LIN {X 0,Y 232.511,Z 383.184,A -85,B 0,C 180,E1 -19720.449,E2 -19720.449} C_VEL
LIN {X 0,Y 232.464,Z 384.387,A -85,B 0,C 180,E1 -19722.217,E2 -19722.217} C_VEL
LIN {X 0,Y 232.571,Z 385.359,A -85,B 0,C 180,E1 -19724.771,E2 -19724.771} C_VEL
LIN {X 0,Y 232.799,Z 385.455,A -85,B 0,C 180,E1 -19727.571,E2 -19727.571} C_VEL
LIN {X 0,Y 233.183,Z 384.978,A -85,B 0,C 180,E1 -19729.361,E2 -19729.361} C_VEL
LIN {X 0,Y 233.739,Z 384.005,A -85,B 0,C 180,E1 -19731.243,E2 -19731.243} C_VEL
LIN {X 0,Y 234.317,Z 382.734,A -85,B 0,C 180,E1 -19732.949,E2 -19732.949} C_VEL
LIN {X 0,Y 235.614,Z 379.876,A -85,B 0,C 180,E1 -19735.626,E2 -19735.626} C_VEL
LIN {X 0,Y 237.292,Z 375.916,A -85,B 0,C 180,E1 -19738.286,E2 -19738.286} C_VEL
LIN {X 0,Y 239.453,Z 370.738,A -85,B 0,C 180,E1 -19740.905,E2 -19740.905} C_VEL
LIN {X 0,Y 241.967,Z 364.116,A -85,B 0,C 180,E1 -19743.494,E2 -19743.494} C_VEL
LIN {X 0,Y 244.993,Z 355.784,A -85,B 0,C 180,E1 -19746.019,E2 -19746.019} C_VEL
LIN {X 0,Y 248.125,Z 346.362,A -85,B 0,C 180,E1 -19748.26,E2 -19748.26} C_VEL
LIN {X 0,Y 250.99,Z 336.548,A -85,B 0,C 180,E1 -19750.091,E2 -19750.091} C_VEL
LIN {X 0,Y 251.249,Z 333.713,A -85,B 0,C 180,E1 -19750.632,E2 -19750.632} C_VEL
LIN {X 0,Y 250.196,Z 324.296,A -85,B 0,C 180,E1 -19752.496,E2 -19752.496} C_VEL
LIN {X 0,Y 248.157,Z 314.273,A -85,B 0,C 180,E1 -19754.352,E2 -19754.352} C_VEL
LIN {X 0,Y 245.125,Z 303.736,A -85,B 0,C 180,E1 -19756.192,E2 -19756.192} C_VEL
LIN {X 0,Y 240.981,Z 293.088,A -85,B 0,C 180,E1 -19758.019,E2 -19758.019} C_VEL
LIN {X 0,Y 237.615,Z 286.034,A -85,B 0,C 180,E1 -19759.239,E2 -19759.239} C_VEL
LIN {X 0,Y 236.078,Z 283.158,A -85,B 0,C 180,E1 -19759.756,E2 -19759.756} C_VEL
LIN {X 0,Y 235.799,Z 281.871,A -85,B 0,C 180,E1 -19759.944,E2 -19759.944} C_VEL
LIN {X 0,Y 235.684,Z 279.573,A -85,B 0,C 180,E1 -19763.621,E2 -19763.621} C_VEL
LIN {X 0,Y 235.395,Z 277.379,A -85,B 0,C 180,E1 -19767.495,E2 -19767.495} C_VEL
LIN {X 0,Y 235.12,Z 275.354,A -85,B 0,C 180,E1 -19771.431,E2 -19771.431} C_VEL
LIN {X 0,Y 234.989,Z 274.23,A -85,B 0,C 180,E1 -19773.794,E2 -19773.794} C_VEL
LIN {X 0,Y 235.036,Z 274.205,A -85,B 0,C 180,E1 -19778.975,E2 -19778.975} C_VEL
LIN {X 0,Y 235.109,Z 274.195,A -85,B 0,C 180,E1 -19783.045,E2 -19783.045} C_VEL
LIN {X 0,Y 235.106,Z 274.199,A -85,B 0,C 180,E1 -19787.924,E2 -19787.924} C_VEL
LIN {X 0,Y 235.324,Z 274.172,A -85,B 0,C 180,E1 -19791.414,E2 -19791.414} C_VEL
LIN {X 0,Y 235.367,Z 274.166,A -85,B 0,C 180,E1 -19793.142,E2 -19793.142} C_VEL
LIN {X 0,Y 235.59,Z 274.14,A -85,B 0,C 180,E1 -19798.293,E2 -19798.293} C_VEL
LIN {X 0,Y 235.59,Z 274.138,A -85,B 0,C 180,E1 -19801.712,E2 -19801.712} C_VEL
LIN {X 0,Y 235.399,Z 274.164,A -85,B 0,C 180,E1 -19806.861,E2 -19806.861} C_VEL
LIN {X 0,Y 235.234,Z 274.184,A -85,B 0,C 180,E1 -19810.329,E2 -19810.329} C_VEL
LIN {X 0,Y 235.109,Z 274.201,A -85,B 0,C 180,E1 -19815.609,E2 -19815.609} C_VEL
LIN {X 0,Y 235.006,Z 274.216,A -85,B 0,C 180,E1 -19819.208,E2 -19819.208} C_VEL
LIN {X 0,Y 234.95,Z 274.225,A -85,B 0,C 180,E1 -19822.886,E2 -19822.886} C_VEL
LIN {X 0,Y 234.954,Z 274.225,A -85,B 0,C 180,E1 -19826.661,E2 -19826.661} C_VEL
LIN {X 0,Y 234.951,Z 274.386,A -85,B 0,C 180,E1 -19829.837,E2 -19829.837} C_VEL
LIN {X 0,Y 235.421,Z 276.965,A -85,B 0,C 180,E1 -19834.558,E2 -19834.558} C_VEL
LIN {X 0,Y 235.9,Z 279.582,A -85,B 0,C 180,E1 -19838.731,E2 -19838.731} C_VEL
LIN {X 0,Y 236.351,Z 282.705,A -85,B 0,C 180,E1 -19843.153,E2 -19843.153} C_VEL
LIN {X 0,Y 236.928,Z 286.376,A -85,B 0,C 180,E1 -19847.868,E2 -19847.868} C_VEL
LIN {X 0,Y 237.196,Z 289.485,A -85,B 0,C 180,E1 -19851.499,E2 -19851.499} C_VEL
LIN {X 0,Y 237.272,Z 290.986,A -85,B 0,C 180,E1 -19852.337,E2 -19852.337} C_VEL
LIN {X 0,Y 237.343,Z 293.485,A -85,B 0,C 180,E1 -19853.038,E2 -19853.038} C_VEL
LIN {X 0,Y 237.459,Z 298.336,A -85,B 0,C 180,E1 -19853.861,E2 -19853.861} C_VEL
LIN {X 0,Y 238.604,Z 313.774,A -85,B 0,C 180,E1 -19855.558,E2 -19855.558} C_VEL
LIN {X 0,Y 238.921,Z 315.576,A -85,B 0,C 180,E1 -19855.823,E2 -19855.823} C_VEL
LIN {X 0,Y 241.212,Z 326.613,A -85,B 0,C 180,E1 -19857.669,E2 -19857.669} C_VEL
LIN {X 0,Y 242.552,Z 337.882,A -85,B 0,C 180,E1 -19859.696,E2 -19859.696} C_VEL
LIN {X 0,Y 242.79,Z 347.643,A -85,B 0,C 180,E1 -19861.611,E2 -19861.611} C_VEL
LIN {X 0,Y 242.31,Z 353.451,A -85,B 0,C 180,E1 -19862.819,E2 -19862.819} C_VEL
LIN {X 0,Y 239.085,Z 362.778,A -85,B 0,C 180,E1 -19864.772,E2 -19864.772} C_VEL
LIN {X 0,Y 235.788,Z 371.794,A -85,B 0,C 180,E1 -19867.203,E2 -19867.203} C_VEL
LIN {X 0,Y 233.117,Z 379.081,A -85,B 0,C 180,E1 -19869.715,E2 -19869.715} C_VEL
LIN {X 0,Y 230.807,Z 384.952,A -85,B 0,C 180,E1 -19872.273,E2 -19872.273} C_VEL
LIN {X 0,Y 228.783,Z 389.609,A -85,B 0,C 180,E1 -19874.864,E2 -19874.864} C_VEL
LIN {X 0,Y 227.416,Z 393.183,A -85,B 0,C 180,E1 -19877.507,E2 -19877.507} C_VEL
LIN {X 0,Y 226.707,Z 395.036,A -85,B 0,C 180,E1 -19879.281,E2 -19879.281} C_VEL
LIN {X 0,Y 225.835,Z 397.451,A -85,B 0,C 180,E1 -19882.85,E2 -19882.85} C_VEL
LIN {X 0,Y 225.588,Z 398.332,A -85,B 0,C 180,E1 -19886.428,E2 -19886.428} C_VEL
LIN {X 0,Y 225.66,Z 398.156,A -85,B 0,C 180,E1 -19888.215,E2 -19888.215} C_VEL
LIN {X 0,Y 225.758,Z 397.585,A -85,B 0,C 180,E1 -19890,E2 -19890} C_VEL
LIN {X 0,Y 225.693,Z 396.616,A -85,B 0,C 180,E1 -19891.784,E2 -19891.784} C_VEL
LIN {X 0,Y 225.669,Z 394.1,A -85,B 0,C 180,E1 -19894.724,E2 -19894.724} C_VEL
LIN {X 0,Y 225.836,Z 391.102,A -85,B 0,C 180,E1 -19897.151,E2 -19897.151} C_VEL
LIN {X 0,Y 226.28,Z 386.756,A -85,B 0,C 180,E1 -19899.836,E2 -19899.836} C_VEL
LIN {X 0,Y 227.026,Z 381.193,A -85,B 0,C 180,E1 -19902.515,E2 -19902.515} C_VEL
LIN {X 0,Y 228.257,Z 374.239,A -85,B 0,C 180,E1 -19905.171,E2 -19905.171} C_VEL
LIN {X 0,Y 229.94,Z 365.512,A -85,B 0,C 180,E1 -19907.797,E2 -19907.797} C_VEL
LIN {X 0,Y 231.048,Z 358.488,A -85,B 0,C 180,E1 -19909.548,E2 -19909.548} C_VEL
LIN {X 0,Y 232.955,Z 347.829,A -85,B 0,C 180,E1 -19911.689,E2 -19911.689} C_VEL
LIN {X 0,Y 233.808,Z 341.483,A -85,B 0,C 180,E1 -19912.768,E2 -19912.768} C_VEL
LIN {X 0,Y 233.356,Z 330.679,A -85,B 0,C 180,E1 -19914.434,E2 -19914.434} C_VEL
LIN {X 0,Y 232.284,Z 318.675,A -85,B 0,C 180,E1 -19915.952,E2 -19915.952} C_VEL
LIN {X 0,Y 230.552,Z 306.518,A -85,B 0,C 180,E1 -19917.209,E2 -19917.209} C_VEL
LIN {X 0,Y 227.885,Z 293.983,A -85,B 0,C 180,E1 -19918.266,E2 -19918.266} C_VEL
LIN {X 0,Y 227.536,Z 291.964,A -85,B 0,C 180,E1 -19918.428,E2 -19918.428} C_VEL
LIN {X 0,Y 228.68,Z 286.481,A -85,B 0,C 180,E1 -19923.585,E2 -19923.585} C_VEL
LIN {X 0,Y 229.087,Z 284.326,A -85,B 0,C 180,E1 -19925.653,E2 -19925.653} C_VEL
LIN {X 0,Y 229.162,Z 282.142,A -85,B 0,C 180,E1 -19927.832,E2 -19927.832} C_VEL
LIN {X 0,Y 228.391,Z 277.71,A -85,B 0,C 180,E1 -19932.607,E2 -19932.607} C_VEL
LIN {X 0,Y 227.881,Z 275.105,A -85,B 0,C 180,E1 -19935.681,E2 -19935.681} C_VEL
LIN {X 0,Y 227.828,Z 275.111,A -85,B 0,C 180,E1 -19940.46,E2 -19940.46} C_VEL
LIN {X 0,Y 227.865,Z 275.102,A -85,B 0,C 180,E1 -19944.123,E2 -19944.123} C_VEL
LIN {X 0,Y 227.855,Z 275.103,A -85,B 0,C 180,E1 -19948.373,E2 -19948.373} C_VEL
LIN {X 0,Y 227.853,Z 275.103,A -85,B 0,C 180,E1 -19952.439,E2 -19952.439} C_VEL
LIN {X 0,Y 227.893,Z 275.095,A -85,B 0,C 180,E1 -19956.363,E2 -19956.363} C_VEL
LIN {X 0,Y 227.931,Z 275.095,A -85,B 0,C 180,E1 -19960.171,E2 -19960.171} C_VEL
LIN {X 0,Y 228.051,Z 275.076,A -85,B 0,C 180,E1 -19963.895,E2 -19963.895} C_VEL
LIN {X 0,Y 228.068,Z 275.075,A -85,B 0,C 180,E1 -19967.541,E2 -19967.541} C_VEL
LIN {X 0,Y 228.264,Z 275.05,A -85,B 0,C 180,E1 -19971.142,E2 -19971.142} C_VEL
LIN {X 0,Y 228.32,Z 275.044,A -85,B 0,C 180,E1 -19972.925,E2 -19972.925} C_VEL
LIN {X 0,Y 228.549,Z 274.995,A -85,B 0,C 180,E1 -19978.236,E2 -19978.236} C_VEL
LIN {X 0,Y 228.55,Z 275.004,A -85,B 0,C 180,E1 -19981.76,E2 -19981.76} C_VEL
LIN {X 0,Y 228.349,Z 275.04,A -85,B 0,C 180,E1 -19987.069,E2 -19987.069} C_VEL
LIN {X 0,Y 228.153,Z 275.06,A -85,B 0,C 180,E1 -19990.649,E2 -19990.649} C_VEL
LIN {X 0,Y 228.053,Z 275.076,A -85,B 0,C 180,E1 -19994.27,E2 -19994.27} C_VEL
LIN {X 0,Y 227.996,Z 275.082,A -85,B 0,C 180,E1 -19997.951,E2 -19997.951} C_VEL
LIN {X 0,Y 227.923,Z 275.09,A -85,B 0,C 180,E1 -20002.327,E2 -20002.327} C_VEL
LIN {X 0,Y 227.935,Z 275.09,A -85,B 0,C 180,E1 -20006.601,E2 -20006.601} C_VEL
LIN {X 0,Y 227.901,Z 275.089,A -85,B 0,C 180,E1 -20010.294,E2 -20010.294} C_VEL
LIN {X 0,Y 227.881,Z 275.096,A -85,B 0,C 180,E1 -20013.717,E2 -20013.717} C_VEL
LIN {X 0,Y 227.863,Z 275.097,A -85,B 0,C 180,E1 -20018.084,E2 -20018.084} C_VEL
LIN {X 0,Y 227.907,Z 275.091,A -85,B 0,C 180,E1 -20022.717,E2 -20022.717} C_VEL
LIN {X 0,Y 227.808,Z 275.103,A -85,B 0,C 180,E1 -20027.258,E2 -20027.258} C_VEL
LIN {X 0,Y 227.84,Z 275.102,A -85,B 0,C 180,E1 -20031.909,E2 -20031.909} C_VEL
LIN {X 0,Y 227.88,Z 275.1,A -85,B 0,C 180,E1 -20036.281,E2 -20036.281} C_VEL
LIN {X 0,Y 227.89,Z 275.099,A -85,B 0,C 180,E1 -20040.434,E2 -20040.434} C_VEL
LIN {X 0,Y 227.869,Z 275.103,A -85,B 0,C 180,E1 -20044.419,E2 -20044.419} C_VEL
LIN {X 0,Y 227.96,Z 275.126,A -85,B 0,C 180,E1 -20047.113,E2 -20047.113} C_VEL
LIN {X 0,Y 227.616,Z 277.511,A -85,B 0,C 180,E1 -20050.145,E2 -20050.145} C_VEL
LIN {X 0,Y 227.294,Z 281.12,A -85,B 0,C 180,E1 -20054.677,E2 -20054.677} C_VEL
LIN {X 0,Y 230.775,Z 294.117,A -85,B 0,C 180,E1 -20055.843,E2 -20055.843} C_VEL
LIN {X 0,Y 233.292,Z 305.864,A -85,B 0,C 180,E1 -20057.142,E2 -20057.142} C_VEL
LIN {X 0,Y 234.888,Z 316.795,A -85,B 0,C 180,E1 -20058.567,E2 -20058.567} C_VEL
LIN {X 0,Y 235.473,Z 324.331,A -85,B 0,C 180,E1 -20059.684,E2 -20059.684} C_VEL
LIN {X 0,Y 233.643,Z 334.908,A -85,B 0,C 180,E1 -20061.35,E2 -20061.35} C_VEL
LIN {X 0,Y 232.151,Z 343.57,A -85,B 0,C 180,E1 -20063.045,E2 -20063.045} C_VEL
LIN {X 0,Y 230.463,Z 352.528,A -85,B 0,C 180,E1 -20065.189,E2 -20065.189} C_VEL
LIN {X 0,Y 228.831,Z 361.274,A -85,B 0,C 180,E1 -20067.8,E2 -20067.8} C_VEL
LIN {X 0,Y 227.567,Z 368.252,A -85,B 0,C 180,E1 -20070.442,E2 -20070.442} C_VEL
LIN {X 0,Y 226.56,Z 374.651,A -85,B 0,C 180,E1 -20073.557,E2 -20073.557} C_VEL
LIN {X 0,Y 226.106,Z 378.454,A -85,B 0,C 180,E1 -20075.956,E2 -20075.956} C_VEL
LIN {X 0,Y 225.564,Z 382.022,A -85,B 0,C 180,E1 -20078.962,E2 -20078.962} C_VEL
LIN {X 0,Y 225.387,Z 383.598,A -85,B 0,C 180,E1 -20080.783,E2 -20080.783} C_VEL
LIN {X 0,Y 225.386,Z 384.708,A -85,B 0,C 180,E1 -20082.607,E2 -20082.607} C_VEL
LIN {X 0,Y 225.471,Z 385.548,A -85,B 0,C 180,E1 -20084.932,E2 -20084.932} C_VEL
LIN {X 0,Y 225.795,Z 385.622,A -85,B 0,C 180,E1 -20088.134,E2 -20088.134} C_VEL
LIN {X 0,Y 226.731,Z 384.25,A -85,B 0,C 180,E1 -20091.586,E2 -20091.586} C_VEL
LIN {X 0,Y 227.507,Z 382.724,A -85,B 0,C 180,E1 -20093.677,E2 -20093.677} C_VEL
LIN {X 0,Y 228.959,Z 379.765,A -85,B 0,C 180,E1 -20096.428,E2 -20096.428} C_VEL
LIN {X 0,Y 230.774,Z 375.692,A -85,B 0,C 180,E1 -20099.16,E2 -20099.16} C_VEL
LIN {X 0,Y 233.497,Z 369.324,A -85,B 0,C 180,E1 -20102.292,E2 -20102.292} C_VEL
LIN {X 0,Y 236.311,Z 362.316,A -85,B 0,C 180,E1 -20104.924,E2 -20104.924} C_VEL
LIN {X 0,Y 238.952,Z 355.344,A -85,B 0,C 180,E1 -20106.997,E2 -20106.997} C_VEL
LIN {X 0,Y 242.083,Z 346.319,A -85,B 0,C 180,E1 -20109.155,E2 -20109.155} C_VEL
LIN {X 0,Y 244.7,Z 337.791,A -85,B 0,C 180,E1 -20110.797,E2 -20110.797} C_VEL
LIN {X 0,Y 244.869,Z 335.253,A -85,B 0,C 180,E1 -20111.308,E2 -20111.308} C_VEL
LIN {X 0,Y 243.908,Z 325.616,A -85,B 0,C 180,E1 -20113.322,E2 -20113.322} C_VEL
LIN {X 0,Y 241.747,Z 314.782,A -85,B 0,C 180,E1 -20115.439,E2 -20115.439} C_VEL
LIN {X 0,Y 238.549,Z 304.085,A -85,B 0,C 180,E1 -20117.436,E2 -20117.436} C_VEL
LIN {X 0,Y 234.502,Z 293.899,A -85,B 0,C 180,E1 -20119.322,E2 -20119.322} C_VEL
LIN {X 0,Y 232.592,Z 290.047,A -85,B 0,C 180,E1 -20120.063,E2 -20120.063} C_VEL
LIN {X 0,Y 230.784,Z 286.427,A -85,B 0,C 180,E1 -20120.746,E2 -20120.746} C_VEL
LIN {X 0,Y 229.169,Z 283.393,A -85,B 0,C 180,E1 -20121.332,E2 -20121.332} C_VEL
LIN {X 0,Y 228.818,Z 282.124,A -85,B 0,C 180,E1 -20121.543,E2 -20121.543} C_VEL
LIN {X 0,Y 228.525,Z 279.364,A -85,B 0,C 180,E1 -20126.391,E2 -20126.391} C_VEL
LIN {X 0,Y 228.252,Z 277.253,A -85,B 0,C 180,E1 -20130.488,E2 -20130.488} C_VEL
LIN {X 0,Y 227.977,Z 275.452,A -85,B 0,C 180,E1 -20134.434,E2 -20134.434} C_VEL
LIN {X 0,Y 227.999,Z 275.086,A -85,B 0,C 180,E1 -20138.293,E2 -20138.293} C_VEL
LIN {X 0,Y 228.038,Z 275.075,A -85,B 0,C 180,E1 -20142.819,E2 -20142.819} C_VEL
LIN {X 0,Y 228.064,Z 275.077,A -85,B 0,C 180,E1 -20147.545,E2 -20147.545} C_VEL
LIN {X 0,Y 228.261,Z 275.052,A -85,B 0,C 180,E1 -20151.147,E2 -20151.147} C_VEL
LIN {X 0,Y 228.317,Z 275.046,A -85,B 0,C 180,E1 -20152.93,E2 -20152.93} C_VEL
LIN {X 0,Y 228.549,Z 275.016,A -85,B 0,C 180,E1 -20158.24,E2 -20158.24} C_VEL
LIN {X 0,Y 228.549,Z 275.015,A -85,B 0,C 180,E1 -20161.764,E2 -20161.764} C_VEL
LIN {X 0,Y 228.35,Z 275.042,A -85,B 0,C 180,E1 -20167.074,E2 -20167.074} C_VEL
LIN {X 0,Y 228.16,Z 275.066,A -85,B 0,C 180,E1 -20170.653,E2 -20170.653} C_VEL
LIN {X 0,Y 228.059,Z 275.08,A -85,B 0,C 180,E1 -20174.274,E2 -20174.274} C_VEL
LIN {X 0,Y 228.001,Z 275.089,A -85,B 0,C 180,E1 -20177.956,E2 -20177.956} C_VEL
LIN {X 0,Y 227.915,Z 275.102,A -85,B 0,C 180,E1 -20182.323,E2 -20182.323} C_VEL
LIN {X 0,Y 227.931,Z 275.1,A -85,B 0,C 180,E1 -20186.599,E2 -20186.599} C_VEL
LIN {X 0,Y 227.864,Z 275.107,A -85,B 0,C 180,E1 -20187.56,E2 -20187.56} C_VEL
LIN {X 0,Y 228.066,Z 276.286,A -85,B 0,C 180,E1 -20190.366,E2 -20190.366} C_VEL
LIN {X 0,Y 228.42,Z 278.112,A -85,B 0,C 180,E1 -20193.828,E2 -20193.828} C_VEL
LIN {X 0,Y 228.828,Z 280.553,A -85,B 0,C 180,E1 -20197.901,E2 -20197.901} C_VEL
LIN {X 0,Y 229.332,Z 283.544,A -85,B 0,C 180,E1 -20202.394,E2 -20202.394} C_VEL
LIN {X 0,Y 229.924,Z 287.556,A -85,B 0,C 180,E1 -20207.744,E2 -20207.744} C_VEL
LIN {X 0,Y 230.202,Z 290.962,A -85,B 0,C 180,E1 -20211.816,E2 -20211.816} C_VEL
LIN {X 0,Y 231.361,Z 294.432,A -85,B 0,C 180,E1 -20212.347,E2 -20212.347} C_VEL
LIN {X 0,Y 232.509,Z 296.395,A -85,B 0,C 180,E1 -20212.734,E2 -20212.734} C_VEL
LIN {X 0,Y 236.743,Z 307.783,A -85,B 0,C 180,E1 -20214.574,E2 -20214.574} C_VEL
LIN {X 0,Y 238.921,Z 315.576,A -85,B 0,C 180,E1 -20215.823,E2 -20215.823} C_VEL
LIN {X 0,Y 239.435,Z 320.71,A -85,B 0,C 180,E1 -20216.542,E2 -20216.542} C_VEL
LIN {X 0,Y 238.405,Z 329.615,A -85,B 0,C 180,E1 -20217.616,E2 -20217.616} C_VEL
LIN {X 0,Y 237.088,Z 336.477,A -85,B 0,C 180,E1 -20218.53,E2 -20218.53} C_VEL
LIN {X 0,Y 236.499,Z 341.335,A -85,B 0,C 180,E1 -20219.337,E2 -20219.337} C_VEL
LIN {X 0,Y 236.473,Z 342.85,A -85,B 0,C 180,E1 -20219.636,E2 -20219.636} C_VEL
LIN {X 0,Y 236.193,Z 352.965,A -85,B 0,C 180,E1 -20221.813,E2 -20221.813} C_VEL
LIN {X 0,Y 234.024,Z 359.687,A -85,B 0,C 180,E1 -20223.227,E2 -20223.227} C_VEL
LIN {X 0,Y 230.92,Z 367.846,A -85,B 0,C 180,E1 -20225.262,E2 -20225.262} C_VEL
LIN {X 0,Y 227.819,Z 375.722,A -85,B 0,C 180,E1 -20227.744,E2 -20227.744} C_VEL
LIN {X 0,Y 225.604,Z 381.322,A -85,B 0,C 180,E1 -20229.961,E2 -20229.961} C_VEL
LIN {X 0,Y 223.256,Z 386.696,A -85,B 0,C 180,E1 -20232.6,E2 -20232.6} C_VEL
LIN {X 0,Y 221.326,Z 390.916,A -85,B 0,C 180,E1 -20235.284,E2 -20235.284} C_VEL
LIN {X 0,Y 220.458,Z 393.166,A -85,B 0,C 180,E1 -20237.106,E2 -20237.106} C_VEL
LIN {X 0,Y 219.712,Z 394.964,A -85,B 0,C 180,E1 -20238.935,E2 -20238.935} C_VEL
LIN {X 0,Y 218.792,Z 397.319,A -85,B 0,C 180,E1 -20242.618,E2 -20242.618} C_VEL
LIN {X 0,Y 218.489,Z 398.087,A -85,B 0,C 180,E1 -20245.702,E2 -20245.702} C_VEL
LIN {X 0,Y 218.575,Z 397.915,A -85,B 0,C 180,E1 -20248.158,E2 -20248.158} C_VEL
LIN {X 0,Y 218.671,Z 397.316,A -85,B 0,C 180,E1 -20250,E2 -20250} C_VEL
LIN {X 0,Y 218.589,Z 396.318,A -85,B 0,C 180,E1 -20251.843,E2 -20251.843} C_VEL
LIN {X 0,Y 218.581,Z 394.005,A -85,B 0,C 180,E1 -20254.61,E2 -20254.61} C_VEL
LIN {X 0,Y 218.788,Z 390.687,A -85,B 0,C 180,E1 -20257.382,E2 -20257.382} C_VEL
LIN {X 0,Y 219.269,Z 386.275,A -85,B 0,C 180,E1 -20260.153,E2 -20260.153} C_VEL
LIN {X 0,Y 220.036,Z 380.639,A -85,B 0,C 180,E1 -20262.919,E2 -20262.919} C_VEL
LIN {X 0,Y 221.384,Z 373.593,A -85,B 0,C 180,E1 -20265.654,E2 -20265.654} C_VEL
LIN {X 0,Y 223.125,Z 364.74,A -85,B 0,C 180,E1 -20268.359,E2 -20268.359} C_VEL
LIN {X 0,Y 224.085,Z 358.762,A -85,B 0,C 180,E1 -20269.897,E2 -20269.897} C_VEL
LIN {X 0,Y 225.832,Z 349.17,A -85,B 0,C 180,E1 -20271.928,E2 -20271.928} C_VEL
LIN {X 0,Y 226.917,Z 343.013,A -85,B 0,C 180,E1 -20273.017,E2 -20273.017} C_VEL
LIN {X 0,Y 226.553,Z 331.665,A -85,B 0,C 180,E1 -20274.875,E2 -20274.875} C_VEL
LIN {X 0,Y 225.576,Z 319.872,A -85,B 0,C 180,E1 -20276.461,E2 -20276.461} C_VEL
LIN {X 0,Y 223.926,Z 307.765,A -85,B 0,C 180,E1 -20277.789,E2 -20277.789} C_VEL
LIN {X 0,Y 221.22,Z 294.742,A -85,B 0,C 180,E1 -20278.956,E2 -20278.956} C_VEL
LIN {X 0,Y 220.581,Z 291.788,A -85,B 0,C 180,E1 -20279.206,E2 -20279.206} C_VEL
LIN {X 0,Y 221.383,Z 288.221,A -85,B 0,C 180,E1 -20282.661,E2 -20282.661} C_VEL
LIN {X 0,Y 222.043,Z 284.998,A -85,B 0,C 180,E1 -20285.841,E2 -20285.841} C_VEL
LIN {X 0,Y 222.143,Z 283.177,A -85,B 0,C 180,E1 -20287.724,E2 -20287.724} C_VEL
LIN {X 0,Y 221.501,Z 279.503,A -85,B 0,C 180,E1 -20291.782,E2 -20291.782} C_VEL
LIN {X 0,Y 220.83,Z 275.983,A -85,B 0,C 180,E1 -20295.983,E2 -20295.983} C_VEL
LIN {X 0,Y 220.782,Z 275.989,A -85,B 0,C 180,E1 -20300.456,E2 -20300.456} C_VEL
LIN {X 0,Y 220.826,Z 275.982,A -85,B 0,C 180,E1 -20302.791,E2 -20302.791} C_VEL
LIN {X 0,Y 220.812,Z 275.979,A -85,B 0,C 180,E1 -20307.241,E2 -20307.241} C_VEL
LIN {X 0,Y 220.803,Z 275.978,A -85,B 0,C 180,E1 -20311.479,E2 -20311.479} C_VEL
LIN {X 0,Y 220.846,Z 275.971,A -85,B 0,C 180,E1 -20315.56,E2 -20315.56} C_VEL
LIN {X 0,Y 220.882,Z 275.971,A -85,B 0,C 180,E1 -20319.511,E2 -20319.511} C_VEL
LIN {X 0,Y 221.012,Z 275.952,A -85,B 0,C 180,E1 -20323.368,E2 -20323.368} C_VEL
LIN {X 0,Y 221.064,Z 275.943,A -85,B 0,C 180,E1 -20329.001,E2 -20329.001} C_VEL
LIN {X 0,Y 221.255,Z 275.924,A -85,B 0,C 180,E1 -20332.698,E2 -20332.698} C_VEL
LIN {X 0,Y 221.507,Z 275.871,A -85,B 0,C 180,E1 -20338.18,E2 -20338.18} C_VEL
LIN {X 0,Y 221.508,Z 275.88,A -85,B 0,C 180,E1 -20341.816,E2 -20341.816} C_VEL
LIN {X 0,Y 221.3,Z 275.919,A -85,B 0,C 180,E1 -20347.296,E2 -20347.296} C_VEL
LIN {X 0,Y 221.101,Z 275.939,A -85,B 0,C 180,E1 -20350.992,E2 -20350.992} C_VEL
LIN {X 0,Y 221.008,Z 275.948,A -85,B 0,C 180,E1 -20356.628,E2 -20356.628} C_VEL
LIN {X 0,Y 220.885,Z 275.969,A -85,B 0,C 180,E1 -20360.484,E2 -20360.484} C_VEL
LIN {X 0,Y 220.86,Z 275.967,A -85,B 0,C 180,E1 -20364.433,E2 -20364.433} C_VEL
LIN {X 0,Y 220.829,Z 275.974,A -85,B 0,C 180,E1 -20368.512,E2 -20368.512} C_VEL
LIN {X 0,Y 220.816,Z 275.977,A -85,B 0,C 180,E1 -20372.753,E2 -20372.753} C_VEL
LIN {X 0,Y 220.83,Z 275.973,A -85,B 0,C 180,E1 -20377.286,E2 -20377.286} C_VEL
LIN {X 0,Y 220.851,Z 275.969,A -85,B 0,C 180,E1 -20381.93,E2 -20381.93} C_VEL
LIN {X 0,Y 220.779,Z 275.982,A -85,B 0,C 180,E1 -20385.548,E2 -20385.548} C_VEL
LIN {X 0,Y 220.798,Z 275.982,A -85,B 0,C 180,E1 -20390.462,E2 -20390.462} C_VEL
LIN {X 0,Y 220.815,Z 275.977,A -85,B 0,C 180,E1 -20392.792,E2 -20392.792} C_VEL
LIN {X 0,Y 220.813,Z 275.979,A -85,B 0,C 180,E1 -20397.244,E2 -20397.244} C_VEL
LIN {X 0,Y 220.807,Z 275.979,A -85,B 0,C 180,E1 -20401.483,E2 -20401.483} C_VEL
LIN {X 0,Y 220.84,Z 275.978,A -85,B 0,C 180,E1 -20405.562,E2 -20405.562} C_VEL
LIN {X 0,Y 220.917,Z 276.039,A -85,B 0,C 180,E1 -20407.016,E2 -20407.016} C_VEL
LIN {X 0,Y 220.43,Z 279.415,A -85,B 0,C 180,E1 -20411.408,E2 -20411.408} C_VEL
LIN {X 0,Y 220.298,Z 281.3,A -85,B 0,C 180,E1 -20413.851,E2 -20413.851} C_VEL
LIN {X 0,Y 224.497,Z 296.96,A -85,B 0,C 180,E1 -20415.4,E2 -20415.4} C_VEL
LIN {X 0,Y 226.85,Z 308.464,A -85,B 0,C 180,E1 -20416.772,E2 -20416.772} C_VEL
LIN {X 0,Y 228.236,Z 318.903,A -85,B 0,C 180,E1 -20418.229,E2 -20418.229} C_VEL
LIN {X 0,Y 228.726,Z 324.731,A -85,B 0,C 180,E1 -20419.152,E2 -20419.152} C_VEL
LIN {X 0,Y 226.83,Z 335.274,A -85,B 0,C 180,E1 -20420.863,E2 -20420.863} C_VEL
LIN {X 0,Y 225.146,Z 344.875,A -85,B 0,C 180,E1 -20422.827,E2 -20422.827} C_VEL
LIN {X 0,Y 223.372,Z 353.659,A -85,B 0,C 180,E1 -20425.036,E2 -20425.036} C_VEL
LIN {X 0,Y 222.009,Z 360.89,A -85,B 0,C 180,E1 -20427.278,E2 -20427.278} C_VEL
LIN {X 0,Y 220.612,Z 368.018,A -85,B 0,C 180,E1 -20430,E2 -20430} C_VEL
LIN {X 0,Y 219.651,Z 373.692,A -85,B 0,C 180,E1 -20432.751,E2 -20432.751} C_VEL
LIN {X 0,Y 219.013,Z 378.657,A -85,B 0,C 180,E1 -20435.888,E2 -20435.888} C_VEL
LIN {X 0,Y 218.428,Z 382.484,A -85,B 0,C 180,E1 -20439.257,E2 -20439.257} C_VEL
LIN {X 0,Y 218.271,Z 383.978,A -85,B 0,C 180,E1 -20441.139,E2 -20441.139} C_VEL
LIN {X 0,Y 218.282,Z 385.029,A -85,B 0,C 180,E1 -20443.025,E2 -20443.025} C_VEL
LIN {X 0,Y 218.381,Z 385.739,A -85,B 0,C 180,E1 -20445.112,E2 -20445.112} C_VEL
LIN {X 0,Y 218.49,Z 385.951,A -85,B 0,C 180,E1 -20446.827,E2 -20446.827} C_VEL
LIN {X 0,Y 218.814,Z 385.758,A -85,B 0,C 180,E1 -20448.734,E2 -20448.734} C_VEL
LIN {X 0,Y 219.769,Z 384.479,A -85,B 0,C 180,E1 -20451.976,E2 -20451.976} C_VEL
LIN {X 0,Y 220.729,Z 382.683,A -85,B 0,C 180,E1 -20454.451,E2 -20454.451} C_VEL
LIN {X 0,Y 222.732,Z 378.734,A -85,B 0,C 180,E1 -20457.938,E2 -20457.938} C_VEL
LIN {X 0,Y 225.082,Z 373.767,A -85,B 0,C 180,E1 -20461.01,E2 -20461.01} C_VEL
LIN {X 0,Y 227.712,Z 367.864,A -85,B 0,C 180,E1 -20463.747,E2 -20463.747} C_VEL
LIN {X 0,Y 230.815,Z 360.387,A -85,B 0,C 180,E1 -20466.422,E2 -20466.422} C_VEL
LIN {X 0,Y 233.761,Z 352.744,A -85,B 0,C 180,E1 -20468.589,E2 -20468.589} C_VEL
LIN {X 0,Y 237.016,Z 343.361,A -85,B 0,C 180,E1 -20470.717,E2 -20470.717} C_VEL
LIN {X 0,Y 238.547,Z 338.428,A -85,B 0,C 180,E1 -20471.66,E2 -20471.66} C_VEL
LIN {X 0,Y 238.05,Z 330.485,A -85,B 0,C 180,E1 -20473.44,E2 -20473.44} C_VEL
LIN {X 0,Y 236.549,Z 320.835,A -85,B 0,C 180,E1 -20475.482,E2 -20475.482} C_VEL
LIN {X 0,Y 234.082,Z 310.774,A -85,B 0,C 180,E1 -20477.509,E2 -20477.509} C_VEL
LIN {X 0,Y 230.19,Z 299.404,A -85,B 0,C 180,E1 -20479.753,E2 -20479.753} C_VEL
LIN {X 0,Y 226.034,Z 290.791,A -85,B 0,C 180,E1 -20481.552,E2 -20481.552} C_VEL
LIN {X 0,Y 224.162,Z 287.123,A -85,B 0,C 180,E1 -20482.316,E2 -20482.316} C_VEL
LIN {X 0,Y 222.322,Z 284.357,A -85,B 0,C 180,E1 -20482.991,E2 -20482.991} C_VEL
LIN {X 0,Y 221.731,Z 282.416,A -85,B 0,C 180,E1 -20483.328,E2 -20483.328} C_VEL
LIN {X 0,Y 221.452,Z 280.252,A -85,B 0,C 180,E1 -20487.353,E2 -20487.353} C_VEL
LIN {X 0,Y 221.21,Z 278.217,A -85,B 0,C 180,E1 -20491.542,E2 -20491.542} C_VEL
LIN {X 0,Y 220.933,Z 276.491,A -85,B 0,C 180,E1 -20495.575,E2 -20495.575} C_VEL
LIN {X 0,Y 220.931,Z 275.962,A -85,B 0,C 180,E1 -20497.562,E2 -20497.562} C_VEL
LIN {X 0,Y 220.986,Z 275.952,A -85,B 0,C 180,E1 -20502.566,E2 -20502.566} C_VEL
LIN {X 0,Y 221.003,Z 275.958,A -85,B 0,C 180,E1 -20507.14,E2 -20507.14} C_VEL
LIN {X 0,Y 221.198,Z 275.933,A -85,B 0,C 180,E1 -20510.861,E2 -20510.861} C_VEL
LIN {X 0,Y 221.253,Z 275.927,A -85,B 0,C 180,E1 -20512.703,E2 -20512.703} C_VEL
LIN {X 0,Y 221.507,Z 275.893,A -85,B 0,C 180,E1 -20518.184,E2 -20518.184} C_VEL
LIN {X 0,Y 221.507,Z 275.892,A -85,B 0,C 180,E1 -20521.82,E2 -20521.82} C_VEL
LIN {X 0,Y 221.285,Z 275.921,A -85,B 0,C 180,E1 -20527.301,E2 -20527.301} C_VEL
LIN {X 0,Y 221.109,Z 275.944,A -85,B 0,C 180,E1 -20530.996,E2 -20530.996} C_VEL
LIN {X 0,Y 221.014,Z 275.96,A -85,B 0,C 180,E1 -20536.632,E2 -20536.632} C_VEL
LIN {X 0,Y 220.883,Z 275.977,A -85,B 0,C 180,E1 -20540.489,E2 -20540.489} C_VEL
LIN {X 0,Y 220.855,Z 275.981,A -85,B 0,C 180,E1 -20544.439,E2 -20544.439} C_VEL
LIN {X 0,Y 220.907,Z 276.372,A -85,B 0,C 180,E1 -20547.029,E2 -20547.029} C_VEL
LIN {X 0,Y 221.178,Z 278.178,A -85,B 0,C 180,E1 -20550.917,E2 -20550.917} C_VEL
LIN {X 0,Y 221.555,Z 280.238,A -85,B 0,C 180,E1 -20554.821,E2 -20554.821} C_VEL
LIN {X 0,Y 221.88,Z 281.874,A -85,B 0,C 180,E1 -20557.641,E2 -20557.641} C_VEL
LIN {X 0,Y 222.255,Z 284.431,A -85,B 0,C 180,E1 -20561.612,E2 -20561.612} C_VEL
LIN {X 0,Y 222.755,Z 287.926,A -85,B 0,C 180,E1 -20566.526,E2 -20566.526} C_VEL
LIN {X 0,Y 223.166,Z 290.957,A -85,B 0,C 180,E1 -20570.149,E2 -20570.149} C_VEL
LIN {X 0,Y 224.317,Z 294.058,A -85,B 0,C 180,E1 -20570.642,E2 -20570.642} C_VEL
LIN {X 0,Y 225.801,Z 296.531,A -85,B 0,C 180,E1 -20571.178,E2 -20571.178} C_VEL
LIN {X 0,Y 229.153,Z 304.463,A -85,B 0,C 180,E1 -20572.624,E2 -20572.624} C_VEL
LIN {X 0,Y 232.696,Z 316.012,A -85,B 0,C 180,E1 -20574.636,E2 -20574.636} C_VEL
LIN {X 0,Y 234.972,Z 327.305,A -85,B 0,C 180,E1 -20576.636,E2 -20576.636} C_VEL
LIN {X 0,Y 236.262,Z 338.849,A -85,B 0,C 180,E1 -20578.822,E2 -20578.822} C_VEL
LIN {X 0,Y 236.473,Z 342.85,A -85,B 0,C 180,E1 -20579.636,E2 -20579.636} C_VEL
LIN {X 0,Y 235.895,Z 346.01,A -85,B 0,C 180,E1 -20580.19,E2 -20580.19} C_VEL
LIN {X 0,Y 234.407,Z 349.2,A -85,B 0,C 180,E1 -20580.649,E2 -20580.649} C_VEL
LIN {X 0,Y 229.068,Z 357.351,A -85,B 0,C 180,E1 -20581.843,E2 -20581.843} C_VEL
LIN {X 0,Y 228.063,Z 359.319,A -85,B 0,C 180,E1 -20582.243,E2 -20582.243} C_VEL
LIN {X 0,Y 224.503,Z 368.177,A -85,B 0,C 180,E1 -20584.505,E2 -20584.505} C_VEL
LIN {X 0,Y 221.048,Z 376.463,A -85,B 0,C 180,E1 -20587.228,E2 -20587.228} C_VEL
LIN {X 0,Y 218.127,Z 383.379,A -85,B 0,C 180,E1 -20590.227,E2 -20590.227} C_VEL
LIN {X 0,Y 215.739,Z 388.279,A -85,B 0,C 180,E1 -20592.952,E2 -20592.952} C_VEL
LIN {X 0,Y 213.944,Z 392.081,A -85,B 0,C 180,E1 -20595.737,E2 -20595.737} C_VEL
LIN {X 0,Y 212.734,Z 394.889,A -85,B 0,C 180,E1 -20598.568,E2 -20598.568} C_VEL
LIN {X 0,Y 211.723,Z 397.188,A -85,B 0,C 180,E1 -20602.37,E2 -20602.37} C_VEL
LIN {X 0,Y 211.399,Z 397.925,A -85,B 0,C 180,E1 -20605.855,E2 -20605.855} C_VEL
LIN {X 0,Y 211.473,Z 397.672,A -85,B 0,C 180,E1 -20608.096,E2 -20608.096} C_VEL
LIN {X 0,Y 211.586,Z 397.047,A -85,B 0,C 180,E1 -20610,E2 -20610} C_VEL
LIN {X 0,Y 211.488,Z 396.02,A -85,B 0,C 180,E1 -20611.904,E2 -20611.904} C_VEL
LIN {X 0,Y 211.479,Z 393.962,A -85,B 0,C 180,E1 -20614.432,E2 -20614.432} C_VEL
LIN {X 0,Y 211.712,Z 390.269,A -85,B 0,C 180,E1 -20617.63,E2 -20617.63} C_VEL
LIN {X 0,Y 212.235,Z 385.792,A -85,B 0,C 180,E1 -20620.494,E2 -20620.494} C_VEL
LIN {X 0,Y 213.072,Z 380.085,A -85,B 0,C 180,E1 -20623.349,E2 -20623.349} C_VEL
LIN {X 0,Y 214.525,Z 372.922,A -85,B 0,C 180,E1 -20626.168,E2 -20626.168} C_VEL
LIN {X 0,Y 216.268,Z 363.961,A -85,B 0,C 180,E1 -20628.963,E2 -20628.963} C_VEL
LIN {X 0,Y 217.29,Z 358.378,A -85,B 0,C 180,E1 -20630.424,E2 -20630.424} C_VEL
LIN {X 0,Y 219.274,Z 348.158,A -85,B 0,C 180,E1 -20632.619,E2 -20632.619} C_VEL
LIN {X 0,Y 220.051,Z 343.203,A -85,B 0,C 180,E1 -20633.529,E2 -20633.529} C_VEL
LIN {X 0,Y 219.692,Z 331.703,A -85,B 0,C 180,E1 -20635.488,E2 -20635.488} C_VEL
LIN {X 0,Y 218.808,Z 320.335,A -85,B 0,C 180,E1 -20637.083,E2 -20637.083} C_VEL
LIN {X 0,Y 217.249,Z 308.688,A -85,B 0,C 180,E1 -20638.434,E2 -20638.434} C_VEL
LIN {X 0,Y 214.755,Z 296.536,A -85,B 0,C 180,E1 -20639.607,E2 -20639.607} C_VEL
LIN {X 0,Y 213.65,Z 291.628,A -85,B 0,C 180,E1 -20640.007,E2 -20640.007} C_VEL
LIN {X 0,Y 214.52,Z 287.821,A -85,B 0,C 180,E1 -20643.844,E2 -20643.844} C_VEL
LIN {X 0,Y 215.077,Z 284.632,A -85,B 0,C 180,E1 -20647.158,E2 -20647.158} C_VEL
LIN {X 0,Y 214.557,Z 281.124,A -85,B 0,C 180,E1 -20651.113,E2 -20651.113} C_VEL
LIN {X 0,Y 213.779,Z 276.862,A -85,B 0,C 180,E1 -20656.338,E2 -20656.338} C_VEL
LIN {X 0,Y 213.705,Z 276.869,A -85,B 0,C 180,E1 -20661.327,E2 -20661.327} C_VEL
LIN {X 0,Y 213.754,Z 276.858,A -85,B 0,C 180,E1 -20666.015,E2 -20666.015} C_VEL
LIN {X 0,Y 213.75,Z 276.856,A -85,B 0,C 180,E1 -20670.447,E2 -20670.447} C_VEL
LIN {X 0,Y 213.781,Z 276.854,A -85,B 0,C 180,E1 -20674.697,E2 -20674.697} C_VEL
LIN {X 0,Y 213.802,Z 276.854,A -85,B 0,C 180,E1 -20678.8,E2 -20678.8} C_VEL
LIN {X 0,Y 213.941,Z 276.833,A -85,B 0,C 180,E1 -20682.801,E2 -20682.801} C_VEL
LIN {X 0,Y 213.948,Z 276.834,A -85,B 0,C 180,E1 -20686.704,E2 -20686.704} C_VEL
LIN {X 0,Y 214.139,Z 276.811,A -85,B 0,C 180,E1 -20690.553,E2 -20690.553} C_VEL
LIN {X 0,Y 214.096,Z 276.814,A -85,B 0,C 180,E1 -20694.346,E2 -20694.346} C_VEL
LIN {X 0,Y 214.44,Z 276.75,A -85,B 0,C 180,E1 -20698.12,E2 -20698.12} C_VEL
LIN {X 0,Y 214.55,Z 276.735,A -85,B 0,C 180,E1 -20699.998,E2 -20699.998} C_VEL
LIN {X 0,Y 214.441,Z 276.76,A -85,B 0,C 180,E1 -20701.876,E2 -20701.876} C_VEL
LIN {X 0,Y 214.235,Z 276.8,A -85,B 0,C 180,E1 -20707.538,E2 -20707.538} C_VEL
LIN {X 0,Y 214.017,Z 276.823,A -85,B 0,C 180,E1 -20711.361,E2 -20711.361} C_VEL
LIN {X 0,Y 213.924,Z 276.837,A -85,B 0,C 180,E1 -20715.235,E2 -20715.235} C_VEL
LIN {X 0,Y 213.833,Z 276.848,A -85,B 0,C 180,E1 -20719.185,E2 -20719.185} C_VEL
LIN {X 0,Y 213.84,Z 276.843,A -85,B 0,C 180,E1 -20723.225,E2 -20723.225} C_VEL
LIN {X 0,Y 213.822,Z 276.849,A -85,B 0,C 180,E1 -20727.448,E2 -20727.448} C_VEL
LIN {X 0,Y 213.772,Z 276.853,A -85,B 0,C 180,E1 -20731.734,E2 -20731.734} C_VEL
LIN {X 0,Y 213.746,Z 276.853,A -85,B 0,C 180,E1 -20736.285,E2 -20736.285} C_VEL
LIN {X 0,Y 213.789,Z 276.851,A -85,B 0,C 180,E1 -20741.104,E2 -20741.104} C_VEL
LIN {X 0,Y 213.8,Z 276.85,A -85,B 0,C 180,E1 -20743.684,E2 -20743.684} C_VEL
LIN {X 0,Y 213.705,Z 276.863,A -85,B 0,C 180,E1 -20748.874,E2 -20748.874} C_VEL
LIN {X 0,Y 213.739,Z 276.858,A -85,B 0,C 180,E1 -20753.712,E2 -20753.712} C_VEL
LIN {X 0,Y 213.76,Z 276.859,A -85,B 0,C 180,E1 -20758.262,E2 -20758.262} C_VEL
LIN {X 0,Y 213.777,Z 276.858,A -85,B 0,C 180,E1 -20762.597,E2 -20762.597} C_VEL
LIN {X 0,Y 213.866,Z 276.97,A -85,B 0,C 180,E1 -20766.938,E2 -20766.938} C_VEL
LIN {X 0,Y 213.451,Z 279.828,A -85,B 0,C 180,E1 -20770.777,E2 -20770.777} C_VEL
LIN {X 0,Y 213.308,Z 281.533,A -85,B 0,C 180,E1 -20773.036,E2 -20773.036} C_VEL
LIN {X 0,Y 217.005,Z 294.785,A -85,B 0,C 180,E1 -20774.375,E2 -20774.375} C_VEL
LIN {X 0,Y 219.741,Z 307.348,A -85,B 0,C 180,E1 -20775.903,E2 -20775.903} C_VEL
LIN {X 0,Y 221.235,Z 317.768,A -85,B 0,C 180,E1 -20777.385,E2 -20777.385} C_VEL
LIN {X 0,Y 221.968,Z 325.141,A -85,B 0,C 180,E1 -20778.587,E2 -20778.587} C_VEL
LIN {X 0,Y 219.859,Z 336.805,A -85,B 0,C 180,E1 -20780.571,E2 -20780.571} C_VEL
LIN {X 0,Y 218.435,Z 344.245,A -85,B 0,C 180,E1 -20782.141,E2 -20782.141} C_VEL
LIN {X 0,Y 216.62,Z 353.158,A -85,B 0,C 180,E1 -20784.414,E2 -20784.414} C_VEL
LIN {X 0,Y 214.868,Z 361.854,A -85,B 0,C 180,E1 -20787.188,E2 -20787.188} C_VEL
LIN {X 0,Y 213.517,Z 368.792,A -85,B 0,C 180,E1 -20790,E2 -20790} C_VEL
LIN {X 0,Y 212.524,Z 374.355,A -85,B 0,C 180,E1 -20792.843,E2 -20792.843} C_VEL
LIN {X 0,Y 211.933,Z 378.904,A -85,B 0,C 180,E1 -20795.849,E2 -20795.849} C_VEL
LIN {X 0,Y 211.568,Z 381.048,A -85,B 0,C 180,E1 -20797.635,E2 -20797.635} C_VEL
LIN {X 0,Y 211.297,Z 382.935,A -85,B 0,C 180,E1 -20799.573,E2 -20799.573} C_VEL
LIN {X 0,Y 211.157,Z 384.345,A -85,B 0,C 180,E1 -20801.519,E2 -20801.519} C_VEL
LIN {X 0,Y 211.185,Z 385.351,A -85,B 0,C 180,E1 -20803.471,E2 -20803.471} C_VEL
LIN {X 0,Y 211.306,Z 385.962,A -85,B 0,C 180,E1 -20805.431,E2 -20805.431} C_VEL
LIN {X 0,Y 211.47,Z 386.144,A -85,B 0,C 180,E1 -20807.403,E2 -20807.403} C_VEL
LIN {X 0,Y 211.849,Z 385.893,A -85,B 0,C 180,E1 -20809.374,E2 -20809.374} C_VEL
LIN {X 0,Y 212.795,Z 384.719,A -85,B 0,C 180,E1 -20812.375,E2 -20812.375} C_VEL
LIN {X 0,Y 214.022,Z 382.626,A -85,B 0,C 180,E1 -20815.27,E2 -20815.27} C_VEL
LIN {X 0,Y 215.936,Z 379.038,A -85,B 0,C 180,E1 -20818.512,E2 -20818.512} C_VEL
LIN {X 0,Y 217.897,Z 375.16,A -85,B 0,C 180,E1 -20821.067,E2 -20821.067} C_VEL
LIN {X 0,Y 220.898,Z 368.907,A -85,B 0,C 180,E1 -20824.192,E2 -20824.192} C_VEL
LIN {X 0,Y 223.749,Z 362.556,A -85,B 0,C 180,E1 -20826.64,E2 -20826.64} C_VEL
LIN {X 0,Y 226.841,Z 355.038,A -85,B 0,C 180,E1 -20828.955,E2 -20828.955} C_VEL
LIN {X 0,Y 230.414,Z 345.462,A -85,B 0,C 180,E1 -20831.268,E2 -20831.268} C_VEL
LIN {X 0,Y 231.972,Z 340.907,A -85,B 0,C 180,E1 -20832.189,E2 -20832.189} C_VEL
LIN {X 0,Y 232.223,Z 337.736,A -85,B 0,C 180,E1 -20832.918,E2 -20832.918} C_VEL
LIN {X 0,Y 231.372,Z 328.347,A -85,B 0,C 180,E1 -20835.111,E2 -20835.111} C_VEL
LIN {X 0,Y 229.584,Z 318.493,A -85,B 0,C 180,E1 -20837.279,E2 -20837.279} C_VEL
LIN {X 0,Y 226.814,Z 308.521,A -85,B 0,C 180,E1 -20839.409,E2 -20839.409} C_VEL
LIN {X 0,Y 223.889,Z 300.538,A -85,B 0,C 180,E1 -20841.114,E2 -20841.114} C_VEL
LIN {X 0,Y 219.68,Z 291.959,A -85,B 0,C 180,E1 -20843.087,E2 -20843.087} C_VEL
LIN {X 0,Y 217.7,Z 288.265,A -85,B 0,C 180,E1 -20843.959,E2 -20843.959} C_VEL
LIN {X 0,Y 215.245,Z 284.675,A -85,B 0,C 180,E1 -20844.932,E2 -20844.932} C_VEL
LIN {X 0,Y 214.653,Z 282.705,A -85,B 0,C 180,E1 -20845.279,E2 -20845.279} C_VEL
LIN {X 0,Y 214.318,Z 280.131,A -85,B 0,C 180,E1 -20850.538,E2 -20850.538} C_VEL
LIN {X 0,Y 214.056,Z 278.343,A -85,B 0,C 180,E1 -20854.737,E2 -20854.737} C_VEL
LIN {X 0,Y 213.847,Z 276.845,A -85,B 0,C 180,E1 -20858.81,E2 -20858.81} C_VEL
LIN {X 0,Y 213.963,Z 276.827,A -85,B 0,C 180,E1 -20862.808,E2 -20862.808} C_VEL
LIN {X 0,Y 213.945,Z 276.833,A -85,B 0,C 180,E1 -20866.709,E2 -20866.709} C_VEL
LIN {X 0,Y 214.136,Z 276.812,A -85,B 0,C 180,E1 -20870.557,E2 -20870.557} C_VEL
LIN {X 0,Y 214.095,Z 276.817,A -85,B 0,C 180,E1 -20874.351,E2 -20874.351} C_VEL
LIN {X 0,Y 214.44,Z 276.773,A -85,B 0,C 180,E1 -20878.124,E2 -20878.124} C_VEL
LIN {X 0,Y 214.54,Z 276.759,A -85,B 0,C 180,E1 -20880.002,E2 -20880.002} C_VEL
LIN {X 0,Y 214.44,Z 276.772,A -85,B 0,C 180,E1 -20881.88,E2 -20881.88} C_VEL
LIN {X 0,Y 214.224,Z 276.799,A -85,B 0,C 180,E1 -20887.543,E2 -20887.543} C_VEL
LIN {X 0,Y 214.041,Z 276.823,A -85,B 0,C 180,E1 -20891.364,E2 -20891.364} C_VEL
LIN {X 0,Y 213.929,Z 276.839,A -85,B 0,C 180,E1 -20895.239,E2 -20895.239} C_VEL
LIN {X 0,Y 213.834,Z 276.853,A -85,B 0,C 180,E1 -20899.19,E2 -20899.19} C_VEL
LIN {X 0,Y 213.802,Z 276.86,A -85,B 0,C 180,E1 -20903.234,E2 -20903.234} C_VEL
LIN {X 0,Y 213.878,Z 277.324,A -85,B 0,C 180,E1 -20905.291,E2 -20905.291} C_VEL
LIN {X 0,Y 214.136,Z 279.116,A -85,B 0,C 180,E1 -20909.494,E2 -20909.494} C_VEL
LIN {X 0,Y 214.522,Z 281.267,A -85,B 0,C 180,E1 -20913.847,E2 -20913.847} C_VEL
LIN {X 0,Y 214.997,Z 283.821,A -85,B 0,C 180,E1 -20918.398,E2 -20918.398} C_VEL
LIN {X 0,Y 215.285,Z 285.666,A -85,B 0,C 180,E1 -20921.339,E2 -20921.339} C_VEL
LIN {X 0,Y 215.692,Z 288.714,A -85,B 0,C 180,E1 -20925.797,E2 -20925.797} C_VEL
LIN {X 0,Y 215.957,Z 290.477,A -85,B 0,C 180,E1 -20928.17,E2 -20928.17} C_VEL
LIN {X 0,Y 217.057,Z 293.507,A -85,B 0,C 180,E1 -20928.685,E2 -20928.685} C_VEL
LIN {X 0,Y 218.947,Z 296.419,A -85,B 0,C 180,E1 -20929.416,E2 -20929.416} C_VEL
LIN {X 0,Y 220.713,Z 300.116,A -85,B 0,C 180,E1 -20930.195,E2 -20930.195} C_VEL
LIN {X 0,Y 223.847,Z 307.749,A -85,B 0,C 180,E1 -20931.715,E2 -20931.715} C_VEL
LIN {X 0,Y 226.86,Z 318.083,A -85,B 0,C 180,E1 -20933.658,E2 -20933.658} C_VEL
LIN {X 0,Y 228.895,Z 328.809,A -85,B 0,C 180,E1 -20935.689,E2 -20935.689} C_VEL
LIN {X 0,Y 230.041,Z 340.514,A -85,B 0,C 180,E1 -20938.046,E2 -20938.046} C_VEL
LIN {X 0,Y 230.107,Z 349.456,A -85,B 0,C 180,E1 -20940.006,E2 -20940.006} C_VEL
LIN {X 0,Y 229.734,Z 354.514,A -85,B 0,C 180,E1 -20941.196,E2 -20941.196} C_VEL
LIN {X 0,Y 228.063,Z 359.319,A -85,B 0,C 180,E1 -20942.243,E2 -20942.243} C_VEL
LIN {X 0,Y 225.747,Z 363.517,A -85,B 0,C 180,E1 -20943.144,E2 -20943.144} C_VEL
LIN {X 0,Y 220.564,Z 369.931,A -85,B 0,C 180,E1 -20944.571,E2 -20944.571} C_VEL
LIN {X 0,Y 215.57,Z 375.692,A -85,B 0,C 180,E1 -20946.201,E2 -20946.201} C_VEL
LIN {X 0,Y 213.585,Z 378.855,A -85,B 0,C 180,E1 -20947.4,E2 -20947.4} C_VEL
LIN {X 0,Y 210.577,Z 385.256,A -85,B 0,C 180,E1 -20950.504,E2 -20950.504} C_VEL
LIN {X 0,Y 208.249,Z 389.71,A -85,B 0,C 180,E1 -20953.331,E2 -20953.331} C_VEL
LIN {X 0,Y 206.571,Z 393.113,A -85,B 0,C 180,E1 -20956.223,E2 -20956.223} C_VEL
LIN {X 0,Y 205.117,Z 396.13,A -85,B 0,C 180,E1 -20960.136,E2 -20960.136} C_VEL
LIN {X 0,Y 204.672,Z 397.058,A -85,B 0,C 180,E1 -20962.106,E2 -20962.106} C_VEL
LIN {X 0,Y 204.327,Z 397.705,A -85,B 0,C 180,E1 -20965.956,E2 -20965.956} C_VEL
LIN {X 0,Y 204.374,Z 397.43,A -85,B 0,C 180,E1 -20968.029,E2 -20968.029} C_VEL
LIN {X 0,Y 204.502,Z 396.777,A -85,B 0,C 180,E1 -20970,E2 -20970} C_VEL
LIN {X 0,Y 204.389,Z 395.713,A -85,B 0,C 180,E1 -20971.971,E2 -20971.971} C_VEL
LIN {X 0,Y 204.384,Z 393.898,A -85,B 0,C 180,E1 -20974.265,E2 -20974.265} C_VEL
LIN {X 0,Y 204.658,Z 389.852,A -85,B 0,C 180,E1 -20977.895,E2 -20977.895} C_VEL
LIN {X 0,Y 205.208,Z 385.307,A -85,B 0,C 180,E1 -20980.857,E2 -20980.857} C_VEL
LIN {X 0,Y 206.369,Z 378.387,A -85,B 0,C 180,E1 -20984.294,E2 -20984.294} C_VEL
LIN {X 0,Y 207.925,Z 370.87,A -85,B 0,C 180,E1 -20987.203,E2 -20987.203} C_VEL
LIN {X 0,Y 209.416,Z 363.171,A -85,B 0,C 180,E1 -20989.609,E2 -20989.609} C_VEL
LIN {X 0,Y 211.368,Z 353.831,A -85,B 0,C 180,E1 -20991.966,E2 -20991.966} C_VEL
LIN {X 0,Y 213.141,Z 344.706,A -85,B 0,C 180,E1 -20993.823,E2 -20993.823} C_VEL
LIN {X 0,Y 212.892,Z 332.59,A -85,B 0,C 180,E1 -20995.995,E2 -20995.995} C_VEL
LIN {X 0,Y 212.118,Z 321.536,A -85,B 0,C 180,E1 -20997.636,E2 -20997.636} C_VEL
LIN {X 0,Y 210.668,Z 310.106,A -85,B 0,C 180,E1 -20999.058,E2 -20999.058} C_VEL
LIN {X 0,Y 208.187,Z 297.654,A -85,B 0,C 180,E1 -21000.355,E2 -21000.355} C_VEL
LIN {X 0,Y 206.788,Z 291.392,A -85,B 0,C 180,E1 -21000.919,E2 -21000.919} C_VEL
LIN {X 0,Y 207.728,Z 287.403,A -85,B 0,C 180,E1 -21005.11,E2 -21005.11} C_VEL
LIN {X 0,Y 208.018,Z 285.259,A -85,B 0,C 180,E1 -21007.454,E2 -21007.454} C_VEL
LIN {X 0,Y 207.429,Z 281.562,A -85,B 0,C 180,E1 -21011.804,E2 -21011.804} C_VEL
LIN {X 0,Y 206.714,Z 277.744,A -85,B 0,C 180,E1 -21016.737,E2 -21016.737} C_VEL
LIN {X 0,Y 206.669,Z 277.745,A -85,B 0,C 180,E1 -21022.255,E2 -21022.255} C_VEL
LIN {X 0,Y 206.694,Z 277.739,A -85,B 0,C 180,E1 -21027.039,E2 -21027.039} C_VEL
LIN {X 0,Y 206.709,Z 277.735,A -85,B 0,C 180,E1 -21032.125,E2 -21032.125} C_VEL
LIN {X 0,Y 206.744,Z 277.729,A -85,B 0,C 180,E1 -21036.608,E2 -21036.608} C_VEL
LIN {X 0,Y 206.87,Z 277.713,A -85,B 0,C 180,E1 -21042.194,E2 -21042.194} C_VEL
LIN {X 0,Y 206.891,Z 277.716,A -85,B 0,C 180,E1 -21046.242,E2 -21046.242} C_VEL
LIN {X 0,Y 207.097,Z 277.687,A -85,B 0,C 180,E1 -21050.229,E2 -21050.229} C_VEL
LIN {X 0,Y 207.057,Z 277.691,A -85,B 0,C 180,E1 -21054.153,E2 -21054.153} C_VEL
LIN {X 0,Y 207.377,Z 277.629,A -85,B 0,C 180,E1 -21058.056,E2 -21058.056} C_VEL
LIN {X 0,Y 207.514,Z 277.61,A -85,B 0,C 180,E1 -21059.998,E2 -21059.998} C_VEL
LIN {X 0,Y 207.081,Z 277.687,A -85,B 0,C 180,E1 -21063.89,E2 -21063.89} C_VEL
LIN {X 0,Y 207.173,Z 277.677,A -85,B 0,C 180,E1 -21067.796,E2 -21067.796} C_VEL
LIN {X 0,Y 206.937,Z 277.707,A -85,B 0,C 180,E1 -21071.755,E2 -21071.755} C_VEL
LIN {X 0,Y 206.857,Z 277.713,A -85,B 0,C 180,E1 -21075.769,E2 -21075.769} C_VEL
LIN {X 0,Y 206.777,Z 277.727,A -85,B 0,C 180,E1 -21079.867,E2 -21079.867} C_VEL
LIN {X 0,Y 206.757,Z 277.723,A -85,B 0,C 180,E1 -21084.07,E2 -21084.07} C_VEL
LIN {X 0,Y 206.737,Z 277.729,A -85,B 0,C 180,E1 -21088.417,E2 -21088.417} C_VEL
LIN {X 0,Y 206.701,Z 277.736,A -85,B 0,C 180,E1 -21092.954,E2 -21092.954} C_VEL
LIN {X 0,Y 206.717,Z 277.731,A -85,B 0,C 180,E1 -21097.728,E2 -21097.728} C_VEL
LIN {X 0,Y 206.717,Z 277.729,A -85,B 0,C 180,E1 -21101.588,E2 -21101.588} C_VEL
LIN {X 0,Y 206.653,Z 277.741,A -85,B 0,C 180,E1 -21105.572,E2 -21105.572} C_VEL
LIN {X 0,Y 206.655,Z 277.742,A -85,B 0,C 180,E1 -21109.749,E2 -21109.749} C_VEL
LIN {X 0,Y 206.722,Z 277.737,A -85,B 0,C 180,E1 -21114.694,E2 -21114.694} C_VEL
LIN {X 0,Y 206.696,Z 277.737,A -85,B 0,C 180,E1 -21119.335,E2 -21119.335} C_VEL
LIN {X 0,Y 206.692,Z 277.738,A -85,B 0,C 180,E1 -21123.767,E2 -21123.767} C_VEL
LIN {X 0,Y 206.841,Z 277.863,A -85,B 0,C 180,E1 -21126.779,E2 -21126.779} C_VEL
LIN {X 0,Y 206.293,Z 281.749,A -85,B 0,C 180,E1 -21132.145,E2 -21132.145} C_VEL
LIN {X 0,Y 209.951,Z 294.238,A -85,B 0,C 180,E1 -21133.465,E2 -21133.465} C_VEL
LIN {X 0,Y 212.797,Z 307.112,A -85,B 0,C 180,E1 -21135.093,E2 -21135.093} C_VEL
LIN {X 0,Y 214.457,Z 318.21,A -85,B 0,C 180,E1 -21136.739,E2 -21136.739} C_VEL
LIN {X 0,Y 215.065,Z 326.918,A -85,B 0,C 180,E1 -21138.215,E2 -21138.215} C_VEL
LIN {X 0,Y 212.829,Z 338.313,A -85,B 0,C 180,E1 -21140.257,E2 -21140.257} C_VEL
LIN {X 0,Y 211.102,Z 347.427,A -85,B 0,C 180,E1 -21142.347,E2 -21142.347} C_VEL
LIN {X 0,Y 209.23,Z 355.805,A -85,B 0,C 180,E1 -21144.7,E2 -21144.7} C_VEL
LIN {X 0,Y 207.736,Z 362.754,A -85,B 0,C 180,E1 -21147.091,E2 -21147.091} C_VEL
LIN {X 0,Y 206.421,Z 369.558,A -85,B 0,C 180,E1 -21150,E2 -21150} C_VEL
LIN {X 0,Y 205.403,Z 375.011,A -85,B 0,C 180,E1 -21152.942,E2 -21152.942} C_VEL
LIN {X 0,Y 204.81,Z 379.276,A -85,B 0,C 180,E1 -21155.909,E2 -21155.909} C_VEL
LIN {X 0,Y 204.417,Z 381.555,A -85,B 0,C 180,E1 -21157.904,E2 -21157.904} C_VEL
LIN {X 0,Y 204.16,Z 383.349,A -85,B 0,C 180,E1 -21159.911,E2 -21159.911} C_VEL
LIN {X 0,Y 204.058,Z 384.71,A -85,B 0,C 180,E1 -21161.926,E2 -21161.926} C_VEL
LIN {X 0,Y 204.227,Z 386.123,A -85,B 0,C 180,E1 -21165.527,E2 -21165.527} C_VEL
LIN {X 0,Y 204.469,Z 386.327,A -85,B 0,C 180,E1 -21168.019,E2 -21168.019} C_VEL
LIN {X 0,Y 204.922,Z 386.029,A -85,B 0,C 180,E1 -21170.057,E2 -21170.057} C_VEL
LIN {X 0,Y 205.85,Z 384.954,A -85,B 0,C 180,E1 -21172.814,E2 -21172.814} C_VEL
LIN {X 0,Y 207.331,Z 382.573,A -85,B 0,C 180,E1 -21176.146,E2 -21176.146} C_VEL
LIN {X 0,Y 209.203,Z 379.315,A -85,B 0,C 180,E1 -21179.144,E2 -21179.144} C_VEL
LIN {X 0,Y 211.569,Z 374.896,A -85,B 0,C 180,E1 -21182.106,E2 -21182.106} C_VEL
LIN {X 0,Y 214.836,Z 368.429,A -85,B 0,C 180,E1 -21185.343,E2 -21185.343} C_VEL
LIN {X 0,Y 218.419,Z 360.617,A -85,B 0,C 180,E1 -21188.271,E2 -21188.271} C_VEL
LIN {X 0,Y 222.021,Z 352.175,A -85,B 0,C 180,E1 -21190.724,E2 -21190.724} C_VEL
LIN {X 0,Y 225.66,Z 342.455,A -85,B 0,C 180,E1 -21192.942,E2 -21192.942} C_VEL
LIN {X 0,Y 225.955,Z 340.158,A -85,B 0,C 180,E1 -21193.483,E2 -21193.483} C_VEL
LIN {X 0,Y 225.302,Z 330.713,A -85,B 0,C 180,E1 -21195.843,E2 -21195.843} C_VEL
LIN {X 0,Y 223.721,Z 320.986,A -85,B 0,C 180,E1 -21198.125,E2 -21198.125} C_VEL
LIN {X 0,Y 220.973,Z 310.598,A -85,B 0,C 180,E1 -21200.502,E2 -21200.502} C_VEL
LIN {X 0,Y 218.145,Z 303.158,A -85,B 0,C 180,E1 -21202.26,E2 -21202.26} C_VEL
LIN {X 0,Y 215.122,Z 296.635,A -85,B 0,C 180,E1 -21203.871,E2 -21203.871} C_VEL
LIN {X 0,Y 212.787,Z 292.378,A -85,B 0,C 180,E1 -21204.995,E2 -21204.995} C_VEL
LIN {X 0,Y 210.857,Z 288.844,A -85,B 0,C 180,E1 -21205.922,E2 -21205.922} C_VEL
LIN {X 0,Y 210.025,Z 287.7,A -85,B 0,C 180,E1 -21206.274,E2 -21206.274} C_VEL
LIN {X 0,Y 208.058,Z 284.826,A -85,B 0,C 180,E1 -21207.144,E2 -21207.144} C_VEL
LIN {X 0,Y 207.505,Z 282.978,A -85,B 0,C 180,E1 -21207.505,E2 -21207.505} C_VEL
LIN {X 0,Y 207.277,Z 281.03,A -85,B 0,C 180,E1 -21211.829,E2 -21211.829} C_VEL
LIN {X 0,Y 207.047,Z 279.232,A -85,B 0,C 180,E1 -21216.414,E2 -21216.414} C_VEL
LIN {X 0,Y 206.845,Z 277.974,A -85,B 0,C 180,E1 -21220.14,E2 -21220.14} C_VEL
LIN {X 0,Y 206.878,Z 277.709,A -85,B 0,C 180,E1 -21222.2,E2 -21222.2} C_VEL
LIN {X 0,Y 206.888,Z 277.709,A -85,B 0,C 180,E1 -21226.246,E2 -21226.246} C_VEL
LIN {X 0,Y 207.094,Z 277.688,A -85,B 0,C 180,E1 -21230.233,E2 -21230.233} C_VEL
LIN {X 0,Y 207.056,Z 277.693,A -85,B 0,C 180,E1 -21234.158,E2 -21234.158} C_VEL
LIN {X 0,Y 207.376,Z 277.652,A -85,B 0,C 180,E1 -21238.06,E2 -21238.06} C_VEL
LIN {X 0,Y 207.506,Z 277.636,A -85,B 0,C 180,E1 -21240.002,E2 -21240.002} C_VEL
LIN {X 0,Y 207.377,Z 277.652,A -85,B 0,C 180,E1 -21241.944,E2 -21241.944} C_VEL
LIN {X 0,Y 207.164,Z 277.678,A -85,B 0,C 180,E1 -21247.801,E2 -21247.801} C_VEL
LIN {X 0,Y 206.978,Z 277.702,A -85,B 0,C 180,E1 -21251.758,E2 -21251.758} C_VEL
LIN {X 0,Y 206.863,Z 277.72,A -85,B 0,C 180,E1 -21255.773,E2 -21255.773} C_VEL
LIN {X 0,Y 206.777,Z 277.735,A -85,B 0,C 180,E1 -21259.872,E2 -21259.872} C_VEL
LIN {X 0,Y 206.745,Z 277.823,A -85,B 0,C 180,E1 -21261.96,E2 -21261.96} C_VEL
LIN {X 0,Y 207.02,Z 279.341,A -85,B 0,C 180,E1 -21266.191,E2 -21266.191} C_VEL
LIN {X 0,Y 207.284,Z 281.229,A -85,B 0,C 180,E1 -21270.571,E2 -21270.571} C_VEL
LIN {X 0,Y 207.798,Z 283.805,A -85,B 0,C 180,E1 -21275.739,E2 -21275.739} C_VEL
LIN {X 0,Y 208.166,Z 286.209,A -85,B 0,C 180,E1 -21279.904,E2 -21279.904} C_VEL
LIN {X 0,Y 208.636,Z 289.517,A -85,B 0,C 180,E1 -21285.026,E2 -21285.026} C_VEL
LIN {X 0,Y 208.806,Z 290.399,A -85,B 0,C 180,E1 -21286.011,E2 -21286.011} C_VEL
LIN {X 0,Y 209.899,Z 293.265,A -85,B 0,C 180,E1 -21286.568,E2 -21286.568} C_VEL
LIN {X 0,Y 211.929,Z 296.209,A -85,B 0,C 180,E1 -21287.417,E2 -21287.417} C_VEL
LIN {X 0,Y 213.9,Z 300.102,A -85,B 0,C 180,E1 -21288.346,E2 -21288.346} C_VEL
LIN {X 0,Y 216.982,Z 306.882,A -85,B 0,C 180,E1 -21289.893,E2 -21289.893} C_VEL
LIN {X 0,Y 219.883,Z 315.343,A -85,B 0,C 180,E1 -21291.679,E2 -21291.679} C_VEL
LIN {X 0,Y 222.176,Z 325.771,A -85,B 0,C 180,E1 -21293.769,E2 -21293.769} C_VEL
LIN {X 0,Y 223.427,Z 335.376,A -85,B 0,C 180,E1 -21295.753,E2 -21295.753} C_VEL
LIN {X 0,Y 223.95,Z 345.154,A -85,B 0,C 180,E1 -21297.924,E2 -21297.924} C_VEL
LIN {X 0,Y 223.365,Z 355.027,A -85,B 0,C 180,E1 -21300.294,E2 -21300.294} C_VEL
LIN {X 0,Y 221.852,Z 359.68,A -85,B 0,C 180,E1 -21301.373,E2 -21301.373} C_VEL
LIN {X 0,Y 218.141,Z 368.509,A -85,B 0,C 180,E1 -21303.706,E2 -21303.706} C_VEL
LIN {X 0,Y 215.109,Z 375.361,A -85,B 0,C 180,E1 -21305.999,E2 -21305.999} C_VEL
LIN {X 0,Y 213.585,Z 378.855,A -85,B 0,C 180,E1 -21307.4,E2 -21307.4} C_VEL
LIN {X 0,Y 211.602,Z 381.846,A -85,B 0,C 180,E1 -21308.667,E2 -21308.667} C_VEL
LIN {X 0,Y 206.697,Z 386.215,A -85,B 0,C 180,E1 -21310.708,E2 -21310.708} C_VEL
LIN {X 0,Y 201.969,Z 389.911,A -85,B 0,C 180,E1 -21312.931,E2 -21312.931} C_VEL
LIN {X 0,Y 200.309,Z 391.762,A -85,B 0,C 180,E1 -21314.456,E2 -21314.456} C_VEL
LIN {X 0,Y 198.773,Z 394.748,A -85,B 0,C 180,E1 -21317.753,E2 -21317.753} C_VEL
LIN {X 0,Y 197.62,Z 396.927,A -85,B 0,C 180,E1 -21321.822,E2 -21321.822} C_VEL
LIN {X 0,Y 197.252,Z 397.484,A -85,B 0,C 180,E1 -21325.914,E2 -21325.914} C_VEL
LIN {X 0,Y 197.277,Z 397.186,A -85,B 0,C 180,E1 -21327.959,E2 -21327.959} C_VEL
LIN {X 0,Y 197.419,Z 396.506,A -85,B 0,C 180,E1 -21330,E2 -21330} C_VEL
LIN {X 0,Y 197.294,Z 395.386,A -85,B 0,C 180,E1 -21332.041,E2 -21332.041} C_VEL
LIN {X 0,Y 197.292,Z 393.828,A -85,B 0,C 180,E1 -21334.085,E2 -21334.085} C_VEL
LIN {X 0,Y 197.487,Z 390.681,A -85,B 0,C 180,E1 -21337.155,E2 -21337.155} C_VEL
LIN {X 0,Y 197.965,Z 386.446,A -85,B 0,C 180,E1 -21340.224,E2 -21340.224} C_VEL
LIN {X 0,Y 198.983,Z 379.983,A -85,B 0,C 180,E1 -21343.792,E2 -21343.792} C_VEL
LIN {X 0,Y 200.538,Z 372.919,A -85,B 0,C 180,E1 -21346.805,E2 -21346.805} C_VEL
LIN {X 0,Y 202.38,Z 364.033,A -85,B 0,C 180,E1 -21349.79,E2 -21349.79} C_VEL
LIN {X 0,Y 203.893,Z 356.889,A -85,B 0,C 180,E1 -21351.749,E2 -21351.749} C_VEL
LIN {X 0,Y 206.096,Z 346.059,A -85,B 0,C 180,E1 -21354.155,E2 -21354.155} C_VEL
LIN {X 0,Y 206.256,Z 339.381,A -85,B 0,C 180,E1 -21355.479,E2 -21355.479} C_VEL
LIN {X 0,Y 205.896,Z 327.912,A -85,B 0,C 180,E1 -21357.438,E2 -21357.438} C_VEL
LIN {X 0,Y 204.665,Z 315.234,A -85,B 0,C 180,E1 -21359.246,E2 -21359.246} C_VEL
LIN {X 0,Y 202.57,Z 302.894,A -85,B 0,C 180,E1 -21360.705,E2 -21360.705} C_VEL
LIN {X 0,Y 199.933,Z 291.188,A -85,B 0,C 180,E1 -21361.867,E2 -21361.867} C_VEL
LIN {X 0,Y 200.879,Z 287.053,A -85,B 0,C 180,E1 -21366.417,E2 -21366.417} C_VEL
LIN {X 0,Y 200.79,Z 284.806,A -85,B 0,C 180,E1 -21369.051,E2 -21369.051} C_VEL
LIN {X 0,Y 200.295,Z 281.991,A -85,B 0,C 180,E1 -21372.533,E2 -21372.533} C_VEL
LIN {X 0,Y 199.647,Z 278.624,A -85,B 0,C 180,E1 -21377.052,E2 -21377.052} C_VEL
LIN {X 0,Y 199.598,Z 278.629,A -85,B 0,C 180,E1 -21380.771,E2 -21380.771} C_VEL
LIN {X 0,Y 199.611,Z 278.62,A -85,B 0,C 180,E1 -21385.711,E2 -21385.711} C_VEL
LIN {X 0,Y 199.686,Z 278.611,A -85,B 0,C 180,E1 -21388.132,E2 -21388.132} C_VEL
LIN {X 0,Y 199.643,Z 278.618,A -85,B 0,C 180,E1 -21392.763,E2 -21392.763} C_VEL
LIN {X 0,Y 199.707,Z 278.606,A -85,B 0,C 180,E1 -21397.223,E2 -21397.223} C_VEL
LIN {X 0,Y 199.795,Z 278.595,A -85,B 0,C 180,E1 -21401.756,E2 -21401.756} C_VEL
LIN {X 0,Y 199.831,Z 278.595,A -85,B 0,C 180,E1 -21405.746,E2 -21405.746} C_VEL
LIN {X 0,Y 200.021,Z 278.566,A -85,B 0,C 180,E1 -21409.879,E2 -21409.879} C_VEL
LIN {X 0,Y 200.019,Z 278.57,A -85,B 0,C 180,E1 -21413.947,E2 -21413.947} C_VEL
LIN {X 0,Y 200.316,Z 278.508,A -85,B 0,C 180,E1 -21417.987,E2 -21417.987} C_VEL
LIN {X 0,Y 200.478,Z 278.485,A -85,B 0,C 180,E1 -21419.998,E2 -21419.998} C_VEL
LIN {X 0,Y 200.027,Z 278.566,A -85,B 0,C 180,E1 -21424.027,E2 -21424.027} C_VEL
LIN {X 0,Y 200.114,Z 278.555,A -85,B 0,C 180,E1 -21428.073,E2 -21428.073} C_VEL
LIN {X 0,Y 199.88,Z 278.586,A -85,B 0,C 180,E1 -21432.176,E2 -21432.176} C_VEL
LIN {X 0,Y 199.796,Z 278.59,A -85,B 0,C 180,E1 -21436.342,E2 -21436.342} C_VEL
LIN {X 0,Y 199.693,Z 278.609,A -85,B 0,C 180,E1 -21440.603,E2 -21440.603} C_VEL
LIN {X 0,Y 199.666,Z 278.608,A -85,B 0,C 180,E1 -21444.982,E2 -21444.982} C_VEL
LIN {X 0,Y 199.667,Z 278.606,A -85,B 0,C 180,E1 -21449.52,E2 -21449.52} C_VEL
LIN {X 0,Y 199.656,Z 278.611,A -85,B 0,C 180,E1 -21452.35,E2 -21452.35} C_VEL
LIN {X 0,Y 199.645,Z 278.609,A -85,B 0,C 180,E1 -21456.755,E2 -21456.755} C_VEL
LIN {X 0,Y 199.692,Z 278.609,A -85,B 0,C 180,E1 -21459.305,E2 -21459.305} C_VEL
LIN {X 0,Y 199.655,Z 278.608,A -85,B 0,C 180,E1 -21462.337,E2 -21462.337} C_VEL
LIN {X 0,Y 199.613,Z 278.619,A -85,B 0,C 180,E1 -21465.239,E2 -21465.239} C_VEL
LIN {X 0,Y 199.632,Z 278.619,A -85,B 0,C 180,E1 -21470.756,E2 -21470.756} C_VEL
LIN {X 0,Y 199.624,Z 278.618,A -85,B 0,C 180,E1 -21475.717,E2 -21475.717} C_VEL
LIN {X 0,Y 199.687,Z 278.612,A -85,B 0,C 180,E1 -21478.135,E2 -21478.135} C_VEL
LIN {X 0,Y 199.632,Z 278.619,A -85,B 0,C 180,E1 -21482.764,E2 -21482.764} C_VEL
LIN {X 0,Y 199.831,Z 278.818,A -85,B 0,C 180,E1 -21486.707,E2 -21486.707} C_VEL
LIN {X 0,Y 199.315,Z 281.895,A -85,B 0,C 180,E1 -21491.138,E2 -21491.138} C_VEL
LIN {X 0,Y 203.497,Z 295.95,A -85,B 0,C 180,E1 -21492.774,E2 -21492.774} C_VEL
LIN {X 0,Y 206.009,Z 307.621,A -85,B 0,C 180,E1 -21494.33,E2 -21494.33} C_VEL
LIN {X 0,Y 207.661,Z 318.402,A -85,B 0,C 180,E1 -21496.007,E2 -21496.007} C_VEL
LIN {X 0,Y 208.362,Z 327.285,A -85,B 0,C 180,E1 -21497.583,E2 -21497.583} C_VEL
LIN {X 0,Y 206.063,Z 338.64,A -85,B 0,C 180,E1 -21499.685,E2 -21499.685} C_VEL
LIN {X 0,Y 204.459,Z 346.809,A -85,B 0,C 180,E1 -21501.6,E2 -21501.6} C_VEL
LIN {X 0,Y 202.492,Z 355.345,A -85,B 0,C 180,E1 -21504.023,E2 -21504.023} C_VEL
LIN {X 0,Y 200.594,Z 363.646,A -85,B 0,C 180,E1 -21506.987,E2 -21506.987} C_VEL
LIN {X 0,Y 199.279,Z 370.323,A -85,B 0,C 180,E1 -21510,E2 -21510} C_VEL
LIN {X 0,Y 198.287,Z 375.662,A -85,B 0,C 180,E1 -21513.047,E2 -21513.047} C_VEL
LIN {X 0,Y 197.656,Z 379.828,A -85,B 0,C 180,E1 -21516.123,E2 -21516.123} C_VEL
LIN {X 0,Y 197.269,Z 382.033,A -85,B 0,C 180,E1 -21518.193,E2 -21518.193} C_VEL
LIN {X 0,Y 197.045,Z 383.757,A -85,B 0,C 180,E1 -21520.272,E2 -21520.272} C_VEL
LIN {X 0,Y 196.974,Z 385.073,A -85,B 0,C 180,E1 -21522.361,E2 -21522.361} C_VEL
LIN {X 0,Y 197.164,Z 386.317,A -85,B 0,C 180,E1 -21525.766,E2 -21525.766} C_VEL
LIN {X 0,Y 197.482,Z 386.509,A -85,B 0,C 180,E1 -21528.68,E2 -21528.68} C_VEL
LIN {X 0,Y 198.012,Z 386.166,A -85,B 0,C 180,E1 -21530.788,E2 -21530.788} C_VEL
LIN {X 0,Y 198.892,Z 385.2,A -85,B 0,C 180,E1 -21533.266,E2 -21533.266} C_VEL
LIN {X 0,Y 200.698,Z 382.52,A -85,B 0,C 180,E1 -21537.079,E2 -21537.079} C_VEL
LIN {X 0,Y 202.473,Z 379.61,A -85,B 0,C 180,E1 -21539.805,E2 -21539.805} C_VEL
LIN {X 0,Y 205.317,Z 374.633,A -85,B 0,C 180,E1 -21543.207,E2 -21543.207} C_VEL
LIN {X 0,Y 208.62,Z 368.38,A -85,B 0,C 180,E1 -21546.359,E2 -21546.359} C_VEL
LIN {X 0,Y 212,Z 361.44,A -85,B 0,C 180,E1 -21549.039,E2 -21549.039} C_VEL
LIN {X 0,Y 215.486,Z 353.686,A -85,B 0,C 180,E1 -21551.402,E2 -21551.402} C_VEL
LIN {X 0,Y 219.525,Z 343.629,A -85,B 0,C 180,E1 -21553.812,E2 -21553.812} C_VEL
LIN {X 0,Y 219.496,Z 335.885,A -85,B 0,C 180,E1 -21555.864,E2 -21555.864} C_VEL
LIN {X 0,Y 218.34,Z 326.156,A -85,B 0,C 180,E1 -21558.342,E2 -21558.342} C_VEL
LIN {X 0,Y 216.272,Z 316.649,A -85,B 0,C 180,E1 -21560.683,E2 -21560.683} C_VEL
LIN {X 0,Y 213.914,Z 309.014,A -85,B 0,C 180,E1 -21562.572,E2 -21562.572} C_VEL
LIN {X 0,Y 210.266,Z 300.771,A -85,B 0,C 180,E1 -21564.794,E2 -21564.794} C_VEL
LIN {X 0,Y 208.47,Z 297.314,A -85,B 0,C 180,E1 -21565.769,E2 -21565.769} C_VEL
LIN {X 0,Y 206.101,Z 293.039,A -85,B 0,C 180,E1 -21567.025,E2 -21567.025} C_VEL
LIN {X 0,Y 204.025,Z 289.56,A -85,B 0,C 180,E1 -21568.097,E2 -21568.097} C_VEL
LIN {X 0,Y 203.453,Z 288.468,A -85,B 0,C 180,E1 -21568.397,E2 -21568.397} C_VEL
LIN {X 0,Y 201.358,Z 285.867,A -85,B 0,C 180,E1 -21569.381,E2 -21569.381} C_VEL
LIN {X 0,Y 200.397,Z 283.281,A -85,B 0,C 180,E1 -21570.019,E2 -21570.019} C_VEL
LIN {X 0,Y 200.258,Z 282.122,A -85,B 0,C 180,E1 -21572.859,E2 -21572.859} C_VEL
LIN {X 0,Y 200.05,Z 280.489,A -85,B 0,C 180,E1 -21577.27,E2 -21577.27} C_VEL
LIN {X 0,Y 199.886,Z 279.111,A -85,B 0,C 180,E1 -21581.676,E2 -21581.676} C_VEL
LIN {X 0,Y 199.807,Z 278.596,A -85,B 0,C 180,E1 -21583.659,E2 -21583.659} C_VEL
LIN {X 0,Y 199.868,Z 278.588,A -85,B 0,C 180,E1 -21587.823,E2 -21587.823} C_VEL
LIN {X 0,Y 200.083,Z 278.561,A -85,B 0,C 180,E1 -21591.926,E2 -21591.926} C_VEL
LIN {X 0,Y 200.316,Z 278.532,A -85,B 0,C 180,E1 -21597.992,E2 -21597.992} C_VEL
LIN {X 0,Y 200.471,Z 278.512,A -85,B 0,C 180,E1 -21600.002,E2 -21600.002} C_VEL
LIN {X 0,Y 200.026,Z 278.567,A -85,B 0,C 180,E1 -21604.032,E2 -21604.032} C_VEL
LIN {X 0,Y 200.108,Z 278.557,A -85,B 0,C 180,E1 -21608.078,E2 -21608.078} C_VEL
LIN {X 0,Y 199.911,Z 278.584,A -85,B 0,C 180,E1 -21612.179,E2 -21612.179} C_VEL
LIN {X 0,Y 199.801,Z 278.602,A -85,B 0,C 180,E1 -21616.346,E2 -21616.346} C_VEL
LIN {X 0,Y 199.782,Z 278.605,A -85,B 0,C 180,E1 -21618.46,E2 -21618.46} C_VEL
LIN {X 0,Y 200.002,Z 280.19,A -85,B 0,C 180,E1 -21623.991,E2 -21623.991} C_VEL
LIN {X 0,Y 200.246,Z 281.998,A -85,B 0,C 180,E1 -21628.67,E2 -21628.67} C_VEL
LIN {X 0,Y 200.673,Z 284.481,A -85,B 0,C 180,E1 -21634.083,E2 -21634.083} C_VEL
LIN {X 0,Y 200.911,Z 285.724,A -85,B 0,C 180,E1 -21636.492,E2 -21636.492} C_VEL
LIN {X 0,Y 201.221,Z 287.574,A -85,B 0,C 180,E1 -21639.792,E2 -21639.792} C_VEL
LIN {X 0,Y 201.496,Z 289.959,A -85,B 0,C 180,E1 -21643.493,E2 -21643.493} C_VEL
LIN {X 0,Y 202.7,Z 293.07,A -85,B 0,C 180,E1 -21644.175,E2 -21644.175} C_VEL
LIN {X 0,Y 204.972,Z 296.12,A -85,B 0,C 180,E1 -21645.216,E2 -21645.216} C_VEL
LIN {X 0,Y 206.988,Z 300.093,A -85,B 0,C 180,E1 -21646.27,E2 -21646.27} C_VEL
LIN {X 0,Y 208.102,Z 302.145,A -85,B 0,C 180,E1 -21646.827,E2 -21646.827} C_VEL
LIN {X 0,Y 211.159,Z 308.628,A -85,B 0,C 180,E1 -21648.494,E2 -21648.494} C_VEL
LIN {X 0,Y 213.753,Z 315.813,A -85,B 0,C 180,E1 -21650.187,E2 -21650.187} C_VEL
LIN {X 0,Y 216.099,Z 326.191,A -85,B 0,C 180,E1 -21652.442,E2 -21652.442} C_VEL
LIN {X 0,Y 217.321,Z 336.276,A -85,B 0,C 180,E1 -21654.65,E2 -21654.65} C_VEL
LIN {X 0,Y 217.706,Z 346.604,A -85,B 0,C 180,E1 -21657.073,E2 -21657.073} C_VEL
LIN {X 0,Y 217.085,Z 355.557,A -85,B 0,C 180,E1 -21659.344,E2 -21659.344} C_VEL
LIN {X 0,Y 216.071,Z 359.237,A -85,B 0,C 180,E1 -21660.263,E2 -21660.263} C_VEL
LIN {X 0,Y 212.452,Z 367.372,A -85,B 0,C 180,E1 -21662.412,E2 -21662.412} C_VEL
LIN {X 0,Y 208.747,Z 375.36,A -85,B 0,C 180,E1 -21665.113,E2 -21665.113} C_VEL
LIN {X 0,Y 205.697,Z 381.803,A -85,B 0,C 180,E1 -21667.925,E2 -21667.925} C_VEL
LIN {X 0,Y 203.025,Z 386.954,A -85,B 0,C 180,E1 -21670.801,E2 -21670.801} C_VEL
LIN {X 0,Y 200.309,Z 391.762,A -85,B 0,C 180,E1 -21674.456,E2 -21674.456} C_VEL
LIN {X 0,Y 198.805,Z 393.394,A -85,B 0,C 180,E1 -21676.032,E2 -21676.032} C_VEL
LIN {X 0,Y 194.856,Z 395.437,A -85,B 0,C 180,E1 -21678.615,E2 -21678.615} C_VEL
LIN {X 0,Y 191.829,Z 396.509,A -85,B 0,C 180,E1 -21680.774,E2 -21680.774} C_VEL
LIN {X 0,Y 190.488,Z 397.019,A -85,B 0,C 180,E1 -21682.497,E2 -21682.497} C_VEL
LIN {X 0,Y 190.337,Z 397.102,A -85,B 0,C 180,E1 -21683.088,E2 -21683.088} C_VEL
LIN {X 0,Y 190.146,Z 397.232,A -85,B 0,C 180,E1 -21686.36,E2 -21686.36} C_VEL
LIN {X 0,Y 190.319,Z 396.228,A -85,B 0,C 180,E1 -21690,E2 -21690} C_VEL
LIN {X 0,Y 190.181,Z 393.835,A -85,B 0,C 180,E1 -21693.802,E2 -21693.802} C_VEL
LIN {X 0,Y 190.435,Z 390.256,A -85,B 0,C 180,E1 -21697.421,E2 -21697.421} C_VEL
LIN {X 0,Y 190.957,Z 385.954,A -85,B 0,C 180,E1 -21700.604,E2 -21700.604} C_VEL
LIN {X 0,Y 192.059,Z 379.415,A -85,B 0,C 180,E1 -21704.3,E2 -21704.3} C_VEL
LIN {X 0,Y 193.714,Z 372.229,A -85,B 0,C 180,E1 -21707.416,E2 -21707.416} C_VEL
LIN {X 0,Y 195.336,Z 364.893,A -85,B 0,C 180,E1 -21709.986,E2 -21709.986} C_VEL
LIN {X 0,Y 196.284,Z 360.13,A -85,B 0,C 180,E1 -21711.414,E2 -21711.414} C_VEL
LIN {X 0,Y 198.382,Z 350.794,A -85,B 0,C 180,E1 -21713.764,E2 -21713.764} C_VEL
LIN {X 0,Y 199.486,Z 344.988,A -85,B 0,C 180,E1 -21715.009,E2 -21715.009} C_VEL
LIN {X 0,Y 199.36,Z 333.407,A -85,B 0,C 180,E1 -21717.276,E2 -21717.276} C_VEL
LIN {X 0,Y 198.65,Z 321.748,A -85,B 0,C 180,E1 -21719.167,E2 -21719.167} C_VEL
LIN {X 0,Y 197.103,Z 309.731,A -85,B 0,C 180,E1 -21720.81,E2 -21720.81} C_VEL
LIN {X 0,Y 194.39,Z 296.599,A -85,B 0,C 180,E1 -21722.315,E2 -21722.315} C_VEL
LIN {X 0,Y 193.078,Z 291.021,A -85,B 0,C 180,E1 -21722.868,E2 -21722.868} C_VEL
LIN {X 0,Y 193.685,Z 288.713,A -85,B 0,C 180,E1 -21725.49,E2 -21725.49} C_VEL
LIN {X 0,Y 193.863,Z 286.549,A -85,B 0,C 180,E1 -21728.045,E2 -21728.045} C_VEL
LIN {X 0,Y 193.507,Z 284.338,A -85,B 0,C 180,E1 -21730.823,E2 -21730.823} C_VEL
LIN {X 0,Y 193.087,Z 282.101,A -85,B 0,C 180,E1 -21733.753,E2 -21733.753} C_VEL
LIN {X 0,Y 192.596,Z 279.503,A -85,B 0,C 180,E1 -21737.365,E2 -21737.365} C_VEL
LIN {X 0,Y 192.583,Z 279.498,A -85,B 0,C 180,E1 -21743.402,E2 -21743.402} C_VEL
LIN {X 0,Y 192.606,Z 279.494,A -85,B 0,C 180,E1 -21747.059,E2 -21747.059} C_VEL
LIN {X 0,Y 192.62,Z 279.489,A -85,B 0,C 180,E1 -21751.682,E2 -21751.682} C_VEL
LIN {X 0,Y 192.678,Z 279.48,A -85,B 0,C 180,E1 -21756.342,E2 -21756.342} C_VEL
LIN {X 0,Y 192.731,Z 279.474,A -85,B 0,C 180,E1 -21761.456,E2 -21761.456} C_VEL
LIN {X 0,Y 192.76,Z 279.475,A -85,B 0,C 180,E1 -21765.211,E2 -21765.211} C_VEL
LIN {X 0,Y 192.943,Z 279.446,A -85,B 0,C 180,E1 -21769.564,E2 -21769.564} C_VEL
LIN {X 0,Y 192.981,Z 279.448,A -85,B 0,C 180,E1 -21773.725,E2 -21773.725} C_VEL
LIN {X 0,Y 193.258,Z 279.386,A -85,B 0,C 180,E1 -21777.913,E2 -21777.913} C_VEL
LIN {X 0,Y 193.442,Z 279.36,A -85,B 0,C 180,E1 -21779.998,E2 -21779.998} C_VEL
LIN {X 0,Y 192.974,Z 279.446,A -85,B 0,C 180,E1 -21784.175,E2 -21784.175} C_VEL
LIN {X 0,Y 193.063,Z 279.432,A -85,B 0,C 180,E1 -21788.37,E2 -21788.37} C_VEL
LIN {X 0,Y 192.803,Z 279.467,A -85,B 0,C 180,E1 -21792.631,E2 -21792.631} C_VEL
LIN {X 0,Y 192.75,Z 279.467,A -85,B 0,C 180,E1 -21796.957,E2 -21796.957} C_VEL
LIN {X 0,Y 192.63,Z 279.489,A -85,B 0,C 180,E1 -21801.395,E2 -21801.395} C_VEL
LIN {X 0,Y 192.657,Z 279.479,A -85,B 0,C 180,E1 -21804.222,E2 -21804.222} C_VEL
LIN {X 0,Y 192.643,Z 279.485,A -85,B 0,C 180,E1 -21808.89,E2 -21808.89} C_VEL
LIN {X 0,Y 192.593,Z 279.494,A -85,B 0,C 180,E1 -21813.184,E2 -21813.184} C_VEL
LIN {X 0,Y 192.604,Z 279.489,A -85,B 0,C 180,E1 -21818.336,E2 -21818.336} C_VEL
LIN {X 0,Y 192.591,Z 279.49,A -85,B 0,C 180,E1 -21823.129,E2 -21823.129} C_VEL
LIN {X 0,Y 192.52,Z 279.499,A -85,B 0,C 180,E1 -21826.891,E2 -21826.891} C_VEL
LIN {X 0,Y 192.565,Z 279.496,A -85,B 0,C 180,E1 -21831.652,E2 -21831.652} C_VEL
LIN {X 0,Y 192.589,Z 279.497,A -85,B 0,C 180,E1 -21836.813,E2 -21836.813} C_VEL
LIN {X 0,Y 192.612,Z 279.492,A -85,B 0,C 180,E1 -21841.684,E2 -21841.684} C_VEL
LIN {X 0,Y 192.747,Z 279.605,A -85,B 0,C 180,E1 -21846.354,E2 -21846.354} C_VEL
LIN {X 0,Y 192.376,Z 282.103,A -85,B 0,C 180,E1 -21850.088,E2 -21850.088} C_VEL
LIN {X 0,Y 196.921,Z 297.101,A -85,B 0,C 180,E1 -21851.968,E2 -21851.968} C_VEL
LIN {X 0,Y 199.374,Z 308.81,A -85,B 0,C 180,E1 -21853.621,E2 -21853.621} C_VEL
LIN {X 0,Y 201.053,Z 320.135,A -85,B 0,C 180,E1 -21855.491,E2 -21855.491} C_VEL
LIN {X 0,Y 201.632,Z 327.666,A -85,B 0,C 180,E1 -21856.905,E2 -21856.905} C_VEL
LIN {X 0,Y 199.318,Z 338.966,A -85,B 0,C 180,E1 -21859.075,E2 -21859.075} C_VEL
LIN {X 0,Y 197.44,Z 348.03,A -85,B 0,C 180,E1 -21861.299,E2 -21861.299} C_VEL
LIN {X 0,Y 195.447,Z 356.371,A -85,B 0,C 180,E1 -21863.807,E2 -21863.807} C_VEL
LIN {X 0,Y 193.476,Z 364.536,A -85,B 0,C 180,E1 -21866.877,E2 -21866.877} C_VEL
LIN {X 0,Y 192.145,Z 371.088,A -85,B 0,C 180,E1 -21870,E2 -21870} C_VEL
LIN {X 0,Y 191.168,Z 376.312,A -85,B 0,C 180,E1 -21873.161,E2 -21873.161} C_VEL
LIN {X 0,Y 190.504,Z 380.378,A -85,B 0,C 180,E1 -21876.354,E2 -21876.354} C_VEL
LIN {X 0,Y 190.126,Z 382.489,A -85,B 0,C 180,E1 -21878.503,E2 -21878.503} C_VEL
LIN {X 0,Y 189.93,Z 384.166,A -85,B 0,C 180,E1 -21880.662,E2 -21880.662} C_VEL
LIN {X 0,Y 189.877,Z 385.437,A -85,B 0,C 180,E1 -21882.831,E2 -21882.831} C_VEL
LIN {X 0,Y 190.085,Z 386.506,A -85,B 0,C 180,E1 -21886.004,E2 -21886.004} C_VEL
LIN {X 0,Y 190.542,Z 386.692,A -85,B 0,C 180,E1 -21889.387,E2 -21889.387} C_VEL
LIN {X 0,Y 191.148,Z 386.3,A -85,B 0,C 180,E1 -21891.571,E2 -21891.571} C_VEL
LIN {X 0,Y 191.946,Z 385.446,A -85,B 0,C 180,E1 -21893.75,E2 -21893.75} C_VEL
LIN {X 0,Y 192.907,Z 384.17,A -85,B 0,C 180,E1 -21895.924,E2 -21895.924} C_VEL
LIN {X 0,Y 194.807,Z 381.418,A -85,B 0,C 180,E1 -21899.145,E2 -21899.145} C_VEL
LIN {X 0,Y 197.212,Z 377.573,A -85,B 0,C 180,E1 -21902.312,E2 -21902.312} C_VEL
LIN {X 0,Y 200.205,Z 372.523,A -85,B 0,C 180,E1 -21905.394,E2 -21905.394} C_VEL
LIN {X 0,Y 203.687,Z 366.103,A -85,B 0,C 180,E1 -21908.393,E2 -21908.393} C_VEL
LIN {X 0,Y 207.7,Z 357.967,A -85,B 0,C 180,E1 -21911.285,E2 -21911.285} C_VEL
LIN {X 0,Y 211.452,Z 349.608,A -85,B 0,C 180,E1 -21913.602,E2 -21913.602} C_VEL
LIN {X 0,Y 212.96,Z 345.87,A -85,B 0,C 180,E1 -21914.488,E2 -21914.488} C_VEL
LIN {X 0,Y 213.429,Z 342.857,A -85,B 0,C 180,E1 -21915.299,E2 -21915.299} C_VEL
LIN {X 0,Y 213.135,Z 334.568,A -85,B 0,C 180,E1 -21917.623,E2 -21917.623} C_VEL
LIN {X 0,Y 212.018,Z 326.009,A -85,B 0,C 180,E1 -21919.915,E2 -21919.915} C_VEL
LIN {X 0,Y 209.806,Z 316.245,A -85,B 0,C 180,E1 -21922.486,E2 -21922.486} C_VEL
LIN {X 0,Y 206.912,Z 308.116,A -85,B 0,C 180,E1 -21924.734,E2 -21924.734} C_VEL
LIN {X 0,Y 204.049,Z 302.114,A -85,B 0,C 180,E1 -21926.562,E2 -21926.562} C_VEL
LIN {X 0,Y 201.874,Z 298.036,A -85,B 0,C 180,E1 -21927.863,E2 -21927.863} C_VEL
LIN {X 0,Y 199.558,Z 293.89,A -85,B 0,C 180,E1 -21929.222,E2 -21929.222} C_VEL
LIN {X 0,Y 197.366,Z 290.436,A -85,B 0,C 180,E1 -21930.454,E2 -21930.454} C_VEL
LIN {X 0,Y 196.489,Z 288.883,A -85,B 0,C 180,E1 -21930.966,E2 -21930.966} C_VEL
LIN {X 0,Y 194.143,Z 285.961,A -85,B 0,C 180,E1 -21932.223,E2 -21932.223} C_VEL
LIN {X 0,Y 193.342,Z 283.632,A -85,B 0,C 180,E1 -21932.832,E2 -21932.832} C_VEL
LIN {X 0,Y 193.188,Z 282.327,A -85,B 0,C 180,E1 -21936.414,E2 -21936.414} C_VEL
LIN {X 0,Y 192.978,Z 280.863,A -85,B 0,C 180,E1 -21941.238,E2 -21941.238} C_VEL
LIN {X 0,Y 192.816,Z 279.864,A -85,B 0,C 180,E1 -21945.221,E2 -21945.221} C_VEL
LIN {X 0,Y 192.94,Z 279.451,A -85,B 0,C 180,E1 -21949.569,E2 -21949.569} C_VEL
LIN {X 0,Y 192.979,Z 279.445,A -85,B 0,C 180,E1 -21953.73,E2 -21953.73} C_VEL
LIN {X 0,Y 193.258,Z 279.411,A -85,B 0,C 180,E1 -21957.918,E2 -21957.918} C_VEL
LIN {X 0,Y 193.435,Z 279.388,A -85,B 0,C 180,E1 -21960.002,E2 -21960.002} C_VEL
LIN {X 0,Y 192.973,Z 279.446,A -85,B 0,C 180,E1 -21964.18,E2 -21964.18} C_VEL
LIN {X 0,Y 193.059,Z 279.436,A -85,B 0,C 180,E1 -21968.375,E2 -21968.375} C_VEL
LIN {X 0,Y 192.85,Z 279.466,A -85,B 0,C 180,E1 -21972.633,E2 -21972.633} C_VEL
LIN {X 0,Y 192.768,Z 279.476,A -85,B 0,C 180,E1 -21974.788,E2 -21974.788} C_VEL
LIN {X 0,Y 192.84,Z 280.408,A -85,B 0,C 180,E1 -21979.15,E2 -21979.15} C_VEL
LIN {X 0,Y 193.123,Z 282.051,A -85,B 0,C 180,E1 -21984.528,E2 -21984.528} C_VEL
LIN {X 0,Y 193.376,Z 283.863,A -85,B 0,C 180,E1 -21989.282,E2 -21989.282} C_VEL
LIN {X 0,Y 193.668,Z 285.709,A -85,B 0,C 180,E1 -21993.423,E2 -21993.423} C_VEL
LIN {X 0,Y 194.062,Z 288.034,A -85,B 0,C 180,E1 -21998.003,E2 -21998.003} C_VEL
LIN {X 0,Y 194.35,Z 289.739,A -85,B 0,C 180,E1 -22000.698,E2 -22000.698} C_VEL
LIN {X 0,Y 195.495,Z 292.654,A -85,B 0,C 180,E1 -22001.433,E2 -22001.433} C_VEL
LIN {X 0,Y 197.919,Z 295.971,A -85,B 0,C 180,E1 -22002.693,E2 -22002.693} C_VEL
LIN {X 0,Y 199.971,Z 299.917,A -85,B 0,C 180,E1 -22003.883,E2 -22003.883} C_VEL
LIN {X 0,Y 201.152,Z 301.794,A -85,B 0,C 180,E1 -22004.507,E2 -22004.507} C_VEL
LIN {X 0,Y 204.172,Z 307.961,A -85,B 0,C 180,E1 -22006.294,E2 -22006.294} C_VEL
LIN {X 0,Y 207.191,Z 315.192,A -85,B 0,C 180,E1 -22008.269,E2 -22008.269} C_VEL
LIN {X 0,Y 209.395,Z 323.134,A -85,B 0,C 180,E1 -22010.194,E2 -22010.194} C_VEL
LIN {X 0,Y 210.838,Z 332.153,A -85,B 0,C 180,E1 -22012.295,E2 -22012.295} C_VEL
LIN {X 0,Y 211.505,Z 342.471,A -85,B 0,C 180,E1 -22014.759,E2 -22014.759} C_VEL
LIN {X 0,Y 211.412,Z 350.503,A -85,B 0,C 180,E1 -22016.822,E2 -22016.822} C_VEL
LIN {X 0,Y 210.538,Z 357.943,A -85,B 0,C 180,E1 -22018.842,E2 -22018.842} C_VEL
LIN {X 0,Y 206.902,Z 366.245,A -85,B 0,C 180,E1 -22021.051,E2 -22021.051} C_VEL
LIN {X 0,Y 202.914,Z 374.393,A -85,B 0,C 180,E1 -22023.795,E2 -22023.795} C_VEL
LIN {X 0,Y 199.784,Z 380.725,A -85,B 0,C 180,E1 -22026.553,E2 -22026.553} C_VEL
LIN {X 0,Y 196.332,Z 387.023,A -85,B 0,C 180,E1 -22030.12,E2 -22030.12} C_VEL
LIN {X 0,Y 193.346,Z 391.967,A -85,B 0,C 180,E1 -22034.093,E2 -22034.093} C_VEL
LIN {X 0,Y 191.806,Z 394.677,A -85,B 0,C 180,E1 -22037.3,E2 -22037.3} C_VEL
LIN {X 0,Y 191.085,Z 395.931,A -85,B 0,C 180,E1 -22039.404,E2 -22039.404} C_VEL
LIN {X 0,Y 190.337,Z 397.102,A -85,B 0,C 180,E1 -22043.088,E2 -22043.088} C_VEL
LIN {X 0,Y 189.548,Z 397.299,A -85,B 0,C 180,E1 -22044.853,E2 -22044.853} C_VEL
LIN {X 0,Y 187.931,Z 397.145,A -85,B 0,C 180,E1 -22046.589,E2 -22046.589} C_VEL
LIN {X 0,Y 184.248,Z 395.945,A -85,B 0,C 180,E1 -22050.09,E2 -22050.09} C_VEL
LIN {X 0,Y 183.198,Z 394.923,A -85,B 0,C 180,E1 -22051.903,E2 -22051.903} C_VEL
LIN {X 0,Y 183.097,Z 394.509,A -85,B 0,C 180,E1 -22052.514,E2 -22052.514} C_VEL
LIN {X 0,Y 183.266,Z 391.063,A -85,B 0,C 180,E1 -22056.606,E2 -22056.606} C_VEL
LIN {X 0,Y 183.716,Z 387.069,A -85,B 0,C 180,E1 -22059.912,E2 -22059.912} C_VEL
LIN {X 0,Y 184.716,Z 380.889,A -85,B 0,C 180,E1 -22063.756,E2 -22063.756} C_VEL
LIN {X 0,Y 186.252,Z 374.134,A -85,B 0,C 180,E1 -22067.004,E2 -22067.004} C_VEL
LIN {X 0,Y 188.235,Z 365.925,A -85,B 0,C 180,E1 -22070.132,E2 -22070.132} C_VEL
LIN {X 0,Y 189.373,Z 360.328,A -85,B 0,C 180,E1 -22071.9,E2 -22071.9} C_VEL
LIN {X 0,Y 191.607,Z 350.888,A -85,B 0,C 180,E1 -22074.37,E2 -22074.37} C_VEL
LIN {X 0,Y 192.635,Z 345.09,A -85,B 0,C 180,E1 -22075.673,E2 -22075.673} C_VEL
LIN {X 0,Y 192.651,Z 335.23,A -85,B 0,C 180,E1 -22077.718,E2 -22077.718} C_VEL
LIN {X 0,Y 192.179,Z 325.055,A -85,B 0,C 180,E1 -22079.512,E2 -22079.512} C_VEL
LIN {X 0,Y 191.02,Z 313.912,A -85,B 0,C 180,E1 -22081.191,E2 -22081.191} C_VEL
LIN {X 0,Y 188.777,Z 301.608,A -85,B 0,C 180,E1 -22082.78,E2 -22082.78} C_VEL
LIN {X 0,Y 186.247,Z 290.819,A -85,B 0,C 180,E1 -22083.984,E2 -22083.984} C_VEL
LIN {X 0,Y 186.788,Z 288.29,A -85,B 0,C 180,E1 -22087.013,E2 -22087.013} C_VEL
LIN {X 0,Y 186.442,Z 285.136,A -85,B 0,C 180,E1 -22091.067,E2 -22091.067} C_VEL
LIN {X 0,Y 185.769,Z 281.612,A -85,B 0,C 180,E1 -22095.955,E2 -22095.955} C_VEL
LIN {X 0,Y 185.536,Z 280.382,A -85,B 0,C 180,E1 -22097.945,E2 -22097.945} C_VEL
LIN {X 0,Y 185.502,Z 280.383,A -85,B 0,C 180,E1 -22102.712,E2 -22102.712} C_VEL
LIN {X 0,Y 185.531,Z 280.374,A -85,B 0,C 180,E1 -22107.97,E2 -22107.97} C_VEL
LIN {X 0,Y 185.548,Z 280.367,A -85,B 0,C 180,E1 -22110.593,E2 -22110.593} C_VEL
LIN {X 0,Y 185.581,Z 280.364,A -85,B 0,C 180,E1 -22115.379,E2 -22115.379} C_VEL
LIN {X 0,Y 185.673,Z 280.354,A -85,B 0,C 180,E1 -22121.132,E2 -22121.132} C_VEL
LIN {X 0,Y 185.691,Z 280.357,A -85,B 0,C 180,E1 -22124.634,E2 -22124.634} C_VEL
LIN {X 0,Y 185.887,Z 280.324,A -85,B 0,C 180,E1 -22129.415,E2 -22129.415} C_VEL
LIN {X 0,Y 185.944,Z 280.324,A -85,B 0,C 180,E1 -22133.487,E2 -22133.487} C_VEL
LIN {X 0,Y 186.202,Z 280.264,A -85,B 0,C 180,E1 -22137.834,E2 -22137.834} C_VEL
LIN {X 0,Y 186.405,Z 280.235,A -85,B 0,C 180,E1 -22139.997,E2 -22139.997} C_VEL
LIN {X 0,Y 185.921,Z 280.324,A -85,B 0,C 180,E1 -22144.333,E2 -22144.333} C_VEL
LIN {X 0,Y 186.009,Z 280.31,A -85,B 0,C 180,E1 -22148.69,E2 -22148.69} C_VEL
LIN {X 0,Y 185.728,Z 280.35,A -85,B 0,C 180,E1 -22153.12,E2 -22153.12} C_VEL
LIN {X 0,Y 185.683,Z 280.349,A -85,B 0,C 180,E1 -22157.623,E2 -22157.623} C_VEL
LIN {X 0,Y 185.59,Z 280.362,A -85,B 0,C 180,E1 -22162.249,E2 -22162.249} C_VEL
LIN {X 0,Y 185.556,Z 280.37,A -85,B 0,C 180,E1 -22167.03,E2 -22167.03} C_VEL
LIN {X 0,Y 185.572,Z 280.361,A -85,B 0,C 180,E1 -22169.491,E2 -22169.491} C_VEL
LIN {X 0,Y 185.513,Z 280.374,A -85,B 0,C 180,E1 -22174.625,E2 -22174.625} C_VEL
LIN {X 0,Y 185.56,Z 280.364,A -85,B 0,C 180,E1 -22177.312,E2 -22177.312} C_VEL
LIN {X 0,Y 185.563,Z 280.368,A -85,B 0,C 180,E1 -22180.759,E2 -22180.759} C_VEL
LIN {X 0,Y 185.543,Z 280.369,A -85,B 0,C 180,E1 -22183.973,E2 -22183.973} C_VEL
LIN {X 0,Y 185.478,Z 280.38,A -85,B 0,C 180,E1 -22189.268,E2 -22189.268} C_VEL
LIN {X 0,Y 185.535,Z 280.37,A -85,B 0,C 180,E1 -22192.695,E2 -22192.695} C_VEL
LIN {X 0,Y 185.524,Z 280.376,A -85,B 0,C 180,E1 -22197.972,E2 -22197.972} C_VEL
LIN {X 0,Y 185.505,Z 280.378,A -85,B 0,C 180,E1 -22202.959,E2 -22202.959} C_VEL
LIN {X 0,Y 185.671,Z 280.4,A -85,B 0,C 180,E1 -22205.99,E2 -22205.99} C_VEL
LIN {X 0,Y 185.469,Z 282.524,A -85,B 0,C 180,E1 -22209.024,E2 -22209.024} C_VEL
LIN {X 0,Y 189.687,Z 295.663,A -85,B 0,C 180,E1 -22210.743,E2 -22210.743} C_VEL
LIN {X 0,Y 192.399,Z 307.934,A -85,B 0,C 180,E1 -22212.545,E2 -22212.545} C_VEL
LIN {X 0,Y 194.17,Z 319.48,A -85,B 0,C 180,E1 -22214.51,E2 -22214.51} C_VEL
LIN {X 0,Y 194.744,Z 329.42,A -85,B 0,C 180,E1 -22216.434,E2 -22216.434} C_VEL
LIN {X 0,Y 192.37,Z 340.337,A -85,B 0,C 180,E1 -22218.675,E2 -22218.675} C_VEL
LIN {X 0,Y 190.403,Z 349.212,A -85,B 0,C 180,E1 -22220.975,E2 -22220.975} C_VEL
LIN {X 0,Y 188.393,Z 357.388,A -85,B 0,C 180,E1 -22223.574,E2 -22223.574} C_VEL
LIN {X 0,Y 186.372,Z 365.417,A -85,B 0,C 180,E1 -22226.757,E2 -22226.757} C_VEL
LIN {X 0,Y 185.017,Z 371.826,A -85,B 0,C 180,E1 -22230,E2 -22230} C_VEL
LIN {X 0,Y 184.047,Z 376.921,A -85,B 0,C 180,E1 -22233.283,E2 -22233.283} C_VEL
LIN {X 0,Y 183.358,Z 380.889,A -85,B 0,C 180,E1 -22236.603,E2 -22236.603} C_VEL
LIN {X 0,Y 182.977,Z 382.943,A -85,B 0,C 180,E1 -22238.837,E2 -22238.837} C_VEL
LIN {X 0,Y 182.799,Z 384.574,A -85,B 0,C 180,E1 -22241.083,E2 -22241.083} C_VEL
LIN {X 0,Y 182.801,Z 385.786,A -85,B 0,C 180,E1 -22243.337,E2 -22243.337} C_VEL
LIN {X 0,Y 183.019,Z 386.696,A -85,B 0,C 180,E1 -22246.27,E2 -22246.27} C_VEL
LIN {X 0,Y 183.608,Z 386.875,A -85,B 0,C 180,E1 -22250.15,E2 -22250.15} C_VEL
LIN {X 0,Y 185.02,Z 385.694,A -85,B 0,C 180,E1 -22254.274,E2 -22254.274} C_VEL
LIN {X 0,Y 186.271,Z 384.17,A -85,B 0,C 180,E1 -22256.92,E2 -22256.92} C_VEL
LIN {X 0,Y 188.333,Z 381.359,A -85,B 0,C 180,E1 -22260.208,E2 -22260.208} C_VEL
LIN {X 0,Y 190.982,Z 377.375,A -85,B 0,C 180,E1 -22263.503,E2 -22263.503} C_VEL
LIN {X 0,Y 194.182,Z 372.213,A -85,B 0,C 180,E1 -22266.667,E2 -22266.667} C_VEL
LIN {X 0,Y 197.944,Z 365.627,A -85,B 0,C 180,E1 -22269.723,E2 -22269.723} C_VEL
LIN {X 0,Y 202.189,Z 357.385,A -85,B 0,C 180,E1 -22272.648,E2 -22272.648} C_VEL
LIN {X 0,Y 206.144,Z 348.798,A -85,B 0,C 180,E1 -22275.024,E2 -22275.024} C_VEL
LIN {X 0,Y 206.946,Z 346.857,A -85,B 0,C 180,E1 -22275.492,E2 -22275.492} C_VEL
LIN {X 0,Y 207.286,Z 341.633,A -85,B 0,C 180,E1 -22277.048,E2 -22277.048} C_VEL
LIN {X 0,Y 206.737,Z 332.312,A -85,B 0,C 180,E1 -22279.77,E2 -22279.77} C_VEL
LIN {X 0,Y 205.481,Z 324.468,A -85,B 0,C 180,E1 -22282.004,E2 -22282.004} C_VEL
LIN {X 0,Y 203.68,Z 317.178,A -85,B 0,C 180,E1 -22284.088,E2 -22284.088} C_VEL
LIN {X 0,Y 200.702,Z 309.299,A -85,B 0,C 180,E1 -22286.532,E2 -22286.532} C_VEL
LIN {X 0,Y 197.399,Z 302.679,A -85,B 0,C 180,E1 -22288.803,E2 -22288.803} C_VEL
LIN {X 0,Y 195.294,Z 298.788,A -85,B 0,C 180,E1 -22290.197,E2 -22290.197} C_VEL
LIN {X 0,Y 192.966,Z 294.563,A -85,B 0,C 180,E1 -22291.743,E2 -22291.743} C_VEL
LIN {X 0,Y 190.759,Z 291.453,A -85,B 0,C 180,E1 -22293.101,E2 -22293.101} C_VEL
LIN {X 0,Y 189.785,Z 289.513,A -85,B 0,C 180,E1 -22293.787,E2 -22293.787} C_VEL
LIN {X 0,Y 187.383,Z 286.848,A -85,B 0,C 180,E1 -22295.229,E2 -22295.229} C_VEL
LIN {X 0,Y 186.273,Z 283.976,A -85,B 0,C 180,E1 -22296.149,E2 -22296.149} C_VEL
LIN {X 0,Y 186.063,Z 282.613,A -85,B 0,C 180,E1 -22300.783,E2 -22300.783} C_VEL
LIN {X 0,Y 185.934,Z 281.649,A -85,B 0,C 180,E1 -22304.66,E2 -22304.66} C_VEL
LIN {X 0,Y 185.94,Z 280.719,A -85,B 0,C 180,E1 -22309.326,E2 -22309.326} C_VEL
LIN {X 0,Y 185.977,Z 280.402,A -85,B 0,C 180,E1 -22311.309,E2 -22311.309} C_VEL
LIN {X 0,Y 186.202,Z 280.289,A -85,B 0,C 180,E1 -22317.84,E2 -22317.84} C_VEL
LIN {X 0,Y 186.399,Z 280.265,A -85,B 0,C 180,E1 -22320.003,E2 -22320.003} C_VEL
LIN {X 0,Y 185.92,Z 280.325,A -85,B 0,C 180,E1 -22324.338,E2 -22324.338} C_VEL
LIN {X 0,Y 186.006,Z 280.316,A -85,B 0,C 180,E1 -22328.695,E2 -22328.695} C_VEL
LIN {X 0,Y 185.85,Z 280.801,A -85,B 0,C 180,E1 -22333.117,E2 -22333.117} C_VEL
LIN {X 0,Y 185.932,Z 281.735,A -85,B 0,C 180,E1 -22337.604,E2 -22337.604} C_VEL
LIN {X 0,Y 186.067,Z 282.978,A -85,B 0,C 180,E1 -22342.195,E2 -22342.195} C_VEL
LIN {X 0,Y 186.234,Z 283.913,A -85,B 0,C 180,E1 -22345.085,E2 -22345.085} C_VEL
LIN {X 0,Y 186.46,Z 285.728,A -85,B 0,C 180,E1 -22349.901,E2 -22349.901} C_VEL
LIN {X 0,Y 186.807,Z 287.696,A -85,B 0,C 180,E1 -22354.358,E2 -22354.358} C_VEL
LIN {X 0,Y 187.089,Z 289.274,A -85,B 0,C 180,E1 -22357.36,E2 -22357.36} C_VEL
LIN {X 0,Y 188.255,Z 292.286,A -85,B 0,C 180,E1 -22358.231,E2 -22358.231} C_VEL
LIN {X 0,Y 190.569,Z 295.082,A -85,B 0,C 180,E1 -22359.591,E2 -22359.591} C_VEL
LIN {X 0,Y 193.136,Z 299.914,A -85,B 0,C 180,E1 -22361.268,E2 -22361.268} C_VEL
LIN {X 0,Y 194.255,Z 301.642,A -85,B 0,C 180,E1 -22361.93,E2 -22361.93} C_VEL
LIN {X 0,Y 196.457,Z 305.818,A -85,B 0,C 180,E1 -22363.349,E2 -22363.349} C_VEL
LIN {X 0,Y 199.556,Z 312.376,A -85,B 0,C 180,E1 -22365.424,E2 -22365.424} C_VEL
LIN {X 0,Y 202.551,Z 320.492,A -85,B 0,C 180,E1 -22367.773,E2 -22367.773} C_VEL
LIN {X 0,Y 204.461,Z 329.16,A -85,B 0,C 180,E1 -22370,E2 -22370} C_VEL
LIN {X 0,Y 205.353,Z 338.841,A -85,B 0,C 180,E1 -22372.412,E2 -22372.412} C_VEL
LIN {X 0,Y 205.369,Z 349.436,A -85,B 0,C 180,E1 -22375.22,E2 -22375.22} C_VEL
LIN {X 0,Y 204.682,Z 356.634,A -85,B 0,C 180,E1 -22377.263,E2 -22377.263} C_VEL
LIN {X 0,Y 203.85,Z 360.162,A -85,B 0,C 180,E1 -22378.281,E2 -22378.281} C_VEL
LIN {X 0,Y 200.012,Z 368.073,A -85,B 0,C 180,E1 -22380.533,E2 -22380.533} C_VEL
LIN {X 0,Y 195.963,Z 375.851,A -85,B 0,C 180,E1 -22383.366,E2 -22383.366} C_VEL
LIN {X 0,Y 192.614,Z 382.091,A -85,B 0,C 180,E1 -22386.337,E2 -22386.337} C_VEL
LIN {X 0,Y 189.666,Z 387.087,A -85,B 0,C 180,E1 -22389.39,E2 -22389.39} C_VEL
LIN {X 0,Y 187.142,Z 390.981,A -85,B 0,C 180,E1 -22392.517,E2 -22392.517} C_VEL
LIN {X 0,Y 184.861,Z 394.611,A -85,B 0,C 180,E1 -22396.815,E2 -22396.815} C_VEL
LIN {X 0,Y 184.097,Z 395.832,A -85,B 0,C 180,E1 -22398.996,E2 -22398.996} C_VEL
LIN {X 0,Y 183.222,Z 397.028,A -85,B 0,C 180,E1 -22403.392,E2 -22403.392} C_VEL
LIN {X 0,Y 183.059,Z 396.947,A -85,B 0,C 180,E1 -22406.586,E2 -22406.586} C_VEL
LIN {X 0,Y 183.222,Z 395.935,A -85,B 0,C 180,E1 -22410,E2 -22410} C_VEL
LIN {X 0,Y 183.097,Z 394.509,A -85,B 0,C 180,E1 -22412.514,E2 -22412.514} C_VEL
LIN {X 0,Y 182.412,Z 393.18,A -85,B 0,C 180,E1 -22414.304,E2 -22414.304} C_VEL
LIN {X 0,Y 179.729,Z 390.361,A -85,B 0,C 180,E1 -22417.198,E2 -22417.198} C_VEL
LIN {X 0,Y 177.642,Z 387.627,A -85,B 0,C 180,E1 -22419.513,E2 -22419.513} C_VEL
LIN {X 0,Y 176.972,Z 385.233,A -85,B 0,C 180,E1 -22421.261,E2 -22421.261} C_VEL
LIN {X 0,Y 177.034,Z 384.367,A -85,B 0,C 180,E1 -22421.839,E2 -22421.839} C_VEL
LIN {X 0,Y 178.243,Z 378.204,A -85,B 0,C 180,E1 -22425.435,E2 -22425.435} C_VEL
LIN {X 0,Y 180.079,Z 370.819,A -85,B 0,C 180,E1 -22428.782,E2 -22428.782} C_VEL
LIN {X 0,Y 181.634,Z 364.157,A -85,B 0,C 180,E1 -22431.246,E2 -22431.246} C_VEL
LIN {X 0,Y 184.127,Z 354.13,A -85,B 0,C 180,E1 -22434.224,E2 -22434.224} C_VEL
LIN {X 0,Y 185.8,Z 346.403,A -85,B 0,C 180,E1 -22436.086,E2 -22436.086} C_VEL
LIN {X 0,Y 185.906,Z 335.755,A -85,B 0,C 180,E1 -22438.429,E2 -22438.429} C_VEL
LIN {X 0,Y 185.463,Z 324.356,A -85,B 0,C 180,E1 -22440.527,E2 -22440.527} C_VEL
LIN {X 0,Y 183.989,Z 311.738,A -85,B 0,C 180,E1 -22442.489,E2 -22442.489} C_VEL
LIN {X 0,Y 181.39,Z 298.501,A -85,B 0,C 180,E1 -22444.247,E2 -22444.247} C_VEL
LIN {X 0,Y 179.44,Z 290.601,A -85,B 0,C 180,E1 -22445.179,E2 -22445.179} C_VEL
LIN {X 0,Y 179.762,Z 288.992,A -85,B 0,C 180,E1 -22447.195,E2 -22447.195} C_VEL
LIN {X 0,Y 179.301,Z 285.544,A -85,B 0,C 180,E1 -22451.86,E2 -22451.86} C_VEL
LIN {X 0,Y 178.854,Z 283.363,A -85,B 0,C 180,E1 -22455.015,E2 -22455.015} C_VEL
LIN {X 0,Y 178.479,Z 281.262,A -85,B 0,C 180,E1 -22458.43,E2 -22458.43} C_VEL
LIN {X 0,Y 178.42,Z 281.262,A -85,B 0,C 180,E1 -22463.78,E2 -22463.78} C_VEL
LIN {X 0,Y 178.485,Z 281.254,A -85,B 0,C 180,E1 -22466.543,E2 -22466.543} C_VEL
LIN {X 0,Y 178.444,Z 281.255,A -85,B 0,C 180,E1 -22471.793,E2 -22471.793} C_VEL
LIN {X 0,Y 178.516,Z 281.245,A -85,B 0,C 180,E1 -22474.887,E2 -22474.887} C_VEL
LIN {X 0,Y 178.621,Z 281.233,A -85,B 0,C 180,E1 -22480.783,E2 -22480.783} C_VEL
LIN {X 0,Y 178.655,Z 281.232,A -85,B 0,C 180,E1 -22486.345,E2 -22486.345} C_VEL
LIN {X 0,Y 178.909,Z 281.199,A -85,B 0,C 180,E1 -22490.957,E2 -22490.957} C_VEL
LIN {X 0,Y 179.148,Z 281.142,A -85,B 0,C 180,E1 -22497.749,E2 -22497.749} C_VEL
LIN {X 0,Y 179.368,Z 281.11,A -85,B 0,C 180,E1 -22499.997,E2 -22499.997} C_VEL
LIN {X 0,Y 178.87,Z 281.202,A -85,B 0,C 180,E1 -22504.504,E2 -22504.504} C_VEL
LIN {X 0,Y 178.959,Z 281.188,A -85,B 0,C 180,E1 -22509.035,E2 -22509.035} C_VEL
LIN {X 0,Y 178.654,Z 281.232,A -85,B 0,C 180,E1 -22513.65,E2 -22513.65} C_VEL
LIN {X 0,Y 178.617,Z 281.234,A -85,B 0,C 180,E1 -22519.213,E2 -22519.213} C_VEL
LIN {X 0,Y 178.518,Z 281.242,A -85,B 0,C 180,E1 -22525.115,E2 -22525.115} C_VEL
LIN {X 0,Y 178.516,Z 281.238,A -85,B 0,C 180,E1 -22529.992,E2 -22529.992} C_VEL
LIN {X 0,Y 178.478,Z 281.25,A -85,B 0,C 180,E1 -22534.217,E2 -22534.217} C_VEL
LIN {X 0,Y 178.473,Z 281.252,A -85,B 0,C 180,E1 -22539.05,E2 -22539.05} C_VEL
LIN {X 0,Y 178.492,Z 281.244,A -85,B 0,C 180,E1 -22542.014,E2 -22542.014} C_VEL
LIN {X 0,Y 178.442,Z 281.257,A -85,B 0,C 180,E1 -22545.144,E2 -22545.144} C_VEL
LIN {X 0,Y 178.411,Z 281.255,A -85,B 0,C 180,E1 -22548.452,E2 -22548.452} C_VEL
LIN {X 0,Y 178.456,Z 281.253,A -85,B 0,C 180,E1 -22551.961,E2 -22551.961} C_VEL
LIN {X 0,Y 178.479,Z 281.254,A -85,B 0,C 180,E1 -22556.546,E2 -22556.546} C_VEL
LIN {X 0,Y 178.438,Z 281.258,A -85,B 0,C 180,E1 -22561.795,E2 -22561.795} C_VEL
LIN {X 0,Y 178.609,Z 281.25,A -85,B 0,C 180,E1 -22565.687,E2 -22565.687} C_VEL
LIN {X 0,Y 178.513,Z 282.523,A -85,B 0,C 180,E1 -22567.781,E2 -22567.781} C_VEL
LIN {X 0,Y 179.55,Z 285.753,A -85,B 0,C 180,E1 -22568.201,E2 -22568.201} C_VEL
LIN {X 0,Y 183.549,Z 298.352,A -85,B 0,C 180,E1 -22570.019,E2 -22570.019} C_VEL
LIN {X 0,Y 186.061,Z 310.375,A -85,B 0,C 180,E1 -22571.93,E2 -22571.93} C_VEL
LIN {X 0,Y 187.665,Z 322.109,A -85,B 0,C 180,E1 -22574.098,E2 -22574.098} C_VEL
LIN {X 0,Y 188.108,Z 329.75,A -85,B 0,C 180,E1 -22575.669,E2 -22575.669} C_VEL
LIN {X 0,Y 185.666,Z 340.632,A -85,B 0,C 180,E1 -22577.984,E2 -22577.984} C_VEL
LIN {X 0,Y 183.379,Z 350.385,A -85,B 0,C 180,E1 -22580.626,E2 -22580.626} C_VEL
LIN {X 0,Y 181.334,Z 358.398,A -85,B 0,C 180,E1 -22583.323,E2 -22583.323} C_VEL
LIN {X 0,Y 179.274,Z 366.26,A -85,B 0,C 180,E1 -22586.629,E2 -22586.629} C_VEL
LIN {X 0,Y 177.89,Z 372.521,A -85,B 0,C 180,E1 -22590,E2 -22590} C_VEL
LIN {X 0,Y 176.922,Z 377.511,A -85,B 0,C 180,E1 -22593.416,E2 -22593.416} C_VEL
LIN {X 0,Y 176.202,Z 381.386,A -85,B 0,C 180,E1 -22596.872,E2 -22596.872} C_VEL
LIN {X 0,Y 175.852,Z 383.392,A -85,B 0,C 180,E1 -22599.199,E2 -22599.199} C_VEL
LIN {X 0,Y 175.679,Z 384.98,A -85,B 0,C 180,E1 -22601.538,E2 -22601.538} C_VEL
LIN {X 0,Y 175.727,Z 386.104,A -85,B 0,C 180,E1 -22603.884,E2 -22603.884} C_VEL
LIN {X 0,Y 175.932,Z 386.88,A -85,B 0,C 180,E1 -22606.529,E2 -22606.529} C_VEL
LIN {X 0,Y 176.706,Z 387.047,A -85,B 0,C 180,E1 -22610.974,E2 -22610.974} C_VEL
LIN {X 0,Y 178.114,Z 385.94,A -85,B 0,C 180,E1 -22614.842,E2 -22614.842} C_VEL
LIN {X 0,Y 179.685,Z 384.171,A -85,B 0,C 180,E1 -22617.992,E2 -22617.992} C_VEL
LIN {X 0,Y 182.504,Z 380.491,A -85,B 0,C 180,E1 -22622.098,E2 -22622.098} C_VEL
LIN {X 0,Y 185.923,Z 375.53,A -85,B 0,C 180,E1 -22625.866,E2 -22625.866} C_VEL
LIN {X 0,Y 189.565,Z 369.801,A -85,B 0,C 180,E1 -22629.068,E2 -22629.068} C_VEL
LIN {X 0,Y 193.731,Z 362.546,A -85,B 0,C 180,E1 -22632.153,E2 -22632.153} C_VEL
LIN {X 0,Y 198.463,Z 353.41,A -85,B 0,C 180,E1 -22635.091,E2 -22635.091} C_VEL
LIN {X 0,Y 200.918,Z 347.978,A -85,B 0,C 180,E1 -22636.536,E2 -22636.536} C_VEL
LIN {X 0,Y 201.163,Z 341.075,A -85,B 0,C 180,E1 -22638.747,E2 -22638.747} C_VEL
LIN {X 0,Y 200.764,Z 333.971,A -85,B 0,C 180,E1 -22640.945,E2 -22640.945} C_VEL
LIN {X 0,Y 199.321,Z 324.528,A -85,B 0,C 180,E1 -22643.812,E2 -22643.812} C_VEL
LIN {X 0,Y 196.977,Z 316.416,A -85,B 0,C 180,E1 -22646.428,E2 -22646.428} C_VEL
LIN {X 0,Y 193.338,Z 308.093,A -85,B 0,C 180,E1 -22649.412,E2 -22649.412} C_VEL
LIN {X 0,Y 189.191,Z 300.08,A -85,B 0,C 180,E1 -22652.56,E2 -22652.56} C_VEL
LIN {X 0,Y 186.994,Z 296.358,A -85,B 0,C 180,E1 -22654.171,E2 -22654.171} C_VEL
LIN {X 0,Y 186.215,Z 295.178,A -85,B 0,C 180,E1 -22654.729,E2 -22654.729} C_VEL
LIN {X 0,Y 183.939,Z 291.951,A -85,B 0,C 180,E1 -22656.351,E2 -22656.351} C_VEL
LIN {X 0,Y 183.021,Z 290.045,A -85,B 0,C 180,E1 -22657.123,E2 -22657.123} C_VEL
LIN {X 0,Y 180.417,Z 287.451,A -85,B 0,C 180,E1 -22658.958,E2 -22658.958} C_VEL
LIN {X 0,Y 179.217,Z 284.724,A -85,B 0,C 180,E1 -22660.057,E2 -22660.057} C_VEL
LIN {X 0,Y 179.145,Z 284.364,A -85,B 0,C 180,E1 -22660.307,E2 -22660.307} C_VEL
LIN {X 0,Y 179.022,Z 283.441,A -85,B 0,C 180,E1 -22664.053,E2 -22664.053} C_VEL
LIN {X 0,Y 179.012,Z 282.474,A -85,B 0,C 180,E1 -22668.954,E2 -22668.954} C_VEL
LIN {X 0,Y 179.02,Z 281.906,A -85,B 0,C 180,E1 -22673.239,E2 -22673.239} C_VEL
LIN {X 0,Y 179.396,Z 281.402,A -85,B 0,C 180,E1 -22680.003,E2 -22680.003} C_VEL
LIN {X 0,Y 179.002,Z 281.726,A -85,B 0,C 180,E1 -22686.767,E2 -22686.767} C_VEL
LIN {X 0,Y 179.022,Z 282.251,A -85,B 0,C 180,E1 -22691.323,E2 -22691.323} C_VEL
LIN {X 0,Y 178.955,Z 283.107,A -85,B 0,C 180,E1 -22695.959,E2 -22695.959} C_VEL
LIN {X 0,Y 179.102,Z 284.237,A -85,B 0,C 180,E1 -22700.683,E2 -22700.683} C_VEL
LIN {X 0,Y 179.333,Z 285.774,A -85,B 0,C 180,E1 -22705.665,E2 -22705.665} C_VEL
LIN {X 0,Y 179.568,Z 287.601,A -85,B 0,C 180,E1 -22710.587,E2 -22710.587} C_VEL
LIN {X 0,Y 179.751,Z 288.749,A -85,B 0,C 180,E1 -22713.28,E2 -22713.28} C_VEL
LIN {X 0,Y 181.043,Z 291.914,A -85,B 0,C 180,E1 -22714.429,E2 -22714.429} C_VEL
LIN {X 0,Y 183.417,Z 294.781,A -85,B 0,C 180,E1 -22716.099,E2 -22716.099} C_VEL
LIN {X 0,Y 184.094,Z 295.695,A -85,B 0,C 180,E1 -22716.564,E2 -22716.564} C_VEL
LIN {X 0,Y 186.004,Z 299.5,A -85,B 0,C 180,E1 -22718.048,E2 -22718.048} C_VEL
LIN {X 0,Y 187.555,Z 301.601,A -85,B 0,C 180,E1 -22719.067,E2 -22719.067} C_VEL
LIN {X 0,Y 189.625,Z 305.684,A -85,B 0,C 180,E1 -22720.613,E2 -22720.613} C_VEL
LIN {X 0,Y 190.844,Z 308.183,A -85,B 0,C 180,E1 -22721.522,E2 -22721.522} C_VEL
LIN {X 0,Y 194.33,Z 315.438,A -85,B 0,C 180,E1 -22724.124,E2 -22724.124} C_VEL
LIN {X 0,Y 196.839,Z 322.322,A -85,B 0,C 180,E1 -22726.308,E2 -22726.308} C_VEL
LIN {X 0,Y 198.342,Z 328.517,A -85,B 0,C 180,E1 -22728.085,E2 -22728.085} C_VEL
LIN {X 0,Y 199.355,Z 337.929,A -85,B 0,C 180,E1 -22730.614,E2 -22730.614} C_VEL
LIN {X 0,Y 199.418,Z 347.323,A -85,B 0,C 180,E1 -22733.194,E2 -22733.194} C_VEL
LIN {X 0,Y 198.813,Z 355.315,A -85,B 0,C 180,E1 -22735.557,E2 -22735.557} C_VEL
LIN {X 0,Y 197.809,Z 360.638,A -85,B 0,C 180,E1 -22737.193,E2 -22737.193} C_VEL
LIN {X 0,Y 193.124,Z 369.796,A -85,B 0,C 180,E1 -22739.976,E2 -22739.976} C_VEL
LIN {X 0,Y 188.996,Z 377.178,A -85,B 0,C 180,E1 -22742.902,E2 -22742.902} C_VEL
LIN {X 0,Y 185.016,Z 384.023,A -85,B 0,C 180,E1 -22746.494,E2 -22746.494} C_VEL
LIN {X 0,Y 182.087,Z 388.568,A -85,B 0,C 180,E1 -22749.674,E2 -22749.674} C_VEL
LIN {X 0,Y 180.38,Z 390.978,A -85,B 0,C 180,E1 -22751.839,E2 -22751.839} C_VEL
LIN {X 0,Y 178.968,Z 392.963,A -85,B 0,C 180,E1 -22754.045,E2 -22754.045} C_VEL
LIN {X 0,Y 177.936,Z 394.545,A -85,B 0,C 180,E1 -22756.292,E2 -22756.292} C_VEL
LIN {X 0,Y 177.097,Z 395.718,A -85,B 0,C 180,E1 -22758.556,E2 -22758.556} C_VEL
LIN {X 0,Y 176.151,Z 396.842,A -85,B 0,C 180,E1 -22763.126,E2 -22763.126} C_VEL
LIN {X 0,Y 175.977,Z 396.628,A -85,B 0,C 180,E1 -22766.825,E2 -22766.825} C_VEL
LIN {X 0,Y 176.127,Z 395.63,A -85,B 0,C 180,E1 -22770,E2 -22770} C_VEL
LIN {X 0,Y 176.002,Z 393.722,A -85,B 0,C 180,E1 -22773.319,E2 -22773.319} C_VEL
LIN {X 0,Y 176.209,Z 390.65,A -85,B 0,C 180,E1 -22776.872,E2 -22776.872} C_VEL
LIN {X 0,Y 176.682,Z 386.586,A -85,B 0,C 180,E1 -22780.311,E2 -22780.311} C_VEL
LIN {X 0,Y 177.034,Z 384.367,A -85,B 0,C 180,E1 -22781.839,E2 -22781.839} C_VEL
LIN {X 0,Y 176.864,Z 381.705,A -85,B 0,C 180,E1 -22783.542,E2 -22783.542} C_VEL
LIN {X 0,Y 175.055,Z 376.817,A -85,B 0,C 180,E1 -22786.308,E2 -22786.308} C_VEL
LIN {X 0,Y 173.603,Z 371.359,A -85,B 0,C 180,E1 -22788.993,E2 -22788.993} C_VEL
LIN {X 0,Y 173.975,Z 367.676,A -85,B 0,C 180,E1 -22790.512,E2 -22790.512} C_VEL
LIN {X 0,Y 175.655,Z 360.539,A -85,B 0,C 180,E1 -22793.034,E2 -22793.034} C_VEL
LIN {X 0,Y 178.12,Z 351.039,A -85,B 0,C 180,E1 -22795.723,E2 -22795.723} C_VEL
LIN {X 0,Y 179,Z 346.486,A -85,B 0,C 180,E1 -22796.841,E2 -22796.841} C_VEL
LIN {X 0,Y 179.209,Z 335.334,A -85,B 0,C 180,E1 -22799.393,E2 -22799.393} C_VEL
LIN {X 0,Y 178.766,Z 323.673,A -85,B 0,C 180,E1 -22801.617,E2 -22801.617} C_VEL
LIN {X 0,Y 177.267,Z 311.306,A -85,B 0,C 180,E1 -22803.632,E2 -22803.632} C_VEL
LIN {X 0,Y 174.875,Z 299.102,A -85,B 0,C 180,E1 -22805.352,E2 -22805.352} C_VEL
LIN {X 0,Y 172.637,Z 290.356,A -85,B 0,C 180,E1 -22806.517,E2 -22806.517} C_VEL
LIN {X 0,Y 172.543,Z 288.337,A -85,B 0,C 180,E1 -22809.29,E2 -22809.29} C_VEL
LIN {X 0,Y 171.984,Z 285.099,A -85,B 0,C 180,E1 -22814.001,E2 -22814.001} C_VEL
LIN {X 0,Y 171.413,Z 282.142,A -85,B 0,C 180,E1 -22818.622,E2 -22818.622} C_VEL
LIN {X 0,Y 171.363,Z 282.144,A -85,B 0,C 180,E1 -22822.031,E2 -22822.031} C_VEL
LIN {X 0,Y 171.399,Z 282.136,A -85,B 0,C 180,E1 -22825.091,E2 -22825.091} C_VEL
LIN {X 0,Y 171.409,Z 282.128,A -85,B 0,C 180,E1 -22830.524,E2 -22830.524} C_VEL
LIN {X 0,Y 171.442,Z 282.124,A -85,B 0,C 180,E1 -22835.796,E2 -22835.796} C_VEL
LIN {X 0,Y 171.577,Z 282.11,A -85,B 0,C 180,E1 -22840.869,E2 -22840.869} C_VEL
LIN {X 0,Y 171.573,Z 282.115,A -85,B 0,C 180,E1 -22845.77,E2 -22845.77} C_VEL
LIN {X 0,Y 171.846,Z 282.079,A -85,B 0,C 180,E1 -22850.582,E2 -22850.582} C_VEL
LIN {X 0,Y 171.81,Z 282.076,A -85,B 0,C 180,E1 -22855.305,E2 -22855.305} C_VEL
LIN {X 0,Y 172.331,Z 281.985,A -85,B 0,C 180,E1 -22859.997,E2 -22859.997} C_VEL
LIN {X 0,Y 171.819,Z 282.081,A -85,B 0,C 180,E1 -22864.69,E2 -22864.69} C_VEL
LIN {X 0,Y 171.886,Z 282.067,A -85,B 0,C 180,E1 -22869.41,E2 -22869.41} C_VEL
LIN {X 0,Y 171.571,Z 282.112,A -85,B 0,C 180,E1 -22874.225,E2 -22874.225} C_VEL
LIN {X 0,Y 171.539,Z 282.117,A -85,B 0,C 180,E1 -22879.559,E2 -22879.559} C_VEL
LIN {X 0,Y 171.456,Z 282.125,A -85,B 0,C 180,E1 -22885.609,E2 -22885.609} C_VEL
LIN {X 0,Y 171.435,Z 282.12,A -85,B 0,C 180,E1 -22890.584,E2 -22890.584} C_VEL
LIN {X 0,Y 171.4,Z 282.129,A -85,B 0,C 180,E1 -22895.029,E2 -22895.029} C_VEL
LIN {X 0,Y 171.426,Z 282.129,A -85,B 0,C 180,E1 -22898.837,E2 -22898.837} C_VEL
LIN {X 0,Y 171.375,Z 282.134,A -85,B 0,C 180,E1 -22904.195,E2 -22904.195} C_VEL
LIN {X 0,Y 171.342,Z 282.138,A -85,B 0,C 180,E1 -22908.984,E2 -22908.984} C_VEL
LIN {X 0,Y 171.405,Z 282.131,A -85,B 0,C 180,E1 -22912.046,E2 -22912.046} C_VEL
LIN {X 0,Y 171.397,Z 282.135,A -85,B 0,C 180,E1 -22915.087,E2 -22915.087} C_VEL
LIN {X 0,Y 171.401,Z 282.135,A -85,B 0,C 180,E1 -22920.526,E2 -22920.526} C_VEL
LIN {X 0,Y 171.58,Z 282.24,A -85,B 0,C 180,E1 -22925.597,E2 -22925.597} C_VEL
LIN {X 0,Y 171.61,Z 282.936,A -85,B 0,C 180,E1 -22926.47,E2 -22926.47} C_VEL
LIN {X 0,Y 175.796,Z 295.389,A -85,B 0,C 180,E1 -22928.343,E2 -22928.343} C_VEL
LIN {X 0,Y 178.573,Z 306.324,A -85,B 0,C 180,E1 -22930.154,E2 -22930.154} C_VEL
LIN {X 0,Y 180.394,Z 317.533,A -85,B 0,C 180,E1 -22932.2,E2 -22932.2} C_VEL
LIN {X 0,Y 181.294,Z 327.449,A -85,B 0,C 180,E1 -22934.255,E2 -22934.255} C_VEL
LIN {X 0,Y 181.229,Z 331.378,A -85,B 0,C 180,E1 -22935.113,E2 -22935.113} C_VEL
LIN {X 0,Y 178.63,Z 342.016,A -85,B 0,C 180,E1 -22937.503,E2 -22937.503} C_VEL
LIN {X 0,Y 176.343,Z 351.562,A -85,B 0,C 180,E1 -22940.248,E2 -22940.248} C_VEL
LIN {X 0,Y 174.272,Z 359.403,A -85,B 0,C 180,E1 -22943.051,E2 -22943.051} C_VEL
LIN {X 0,Y 172.169,Z 367.07,A -85,B 0,C 180,E1 -22946.49,E2 -22946.49} C_VEL
LIN {X 0,Y 170.761,Z 373.217,A -85,B 0,C 180,E1 -22950,E2 -22950} C_VEL
LIN {X 0,Y 169.774,Z 378.104,A -85,B 0,C 180,E1 -22953.56,E2 -22953.56} C_VEL
LIN {X 0,Y 169.044,Z 381.883,A -85,B 0,C 180,E1 -22957.165,E2 -22957.165} C_VEL
LIN {X 0,Y 168.713,Z 383.844,A -85,B 0,C 180,E1 -22959.591,E2 -22959.591} C_VEL
LIN {X 0,Y 168.567,Z 385.358,A -85,B 0,C 180,E1 -22962.032,E2 -22962.032} C_VEL
LIN {X 0,Y 168.653,Z 386.421,A -85,B 0,C 180,E1 -22964.479,E2 -22964.479} C_VEL
LIN {X 0,Y 168.874,Z 387.09,A -85,B 0,C 180,E1 -22966.936,E2 -22966.936} C_VEL
LIN {X 0,Y 169.212,Z 387.366,A -85,B 0,C 180,E1 -22969.406,E2 -22969.406} C_VEL
LIN {X 0,Y 169.837,Z 387.187,A -85,B 0,C 180,E1 -22971.865,E2 -22971.865} C_VEL
LIN {X 0,Y 171.233,Z 386.185,A -85,B 0,C 180,E1 -22975.458,E2 -22975.458} C_VEL
LIN {X 0,Y 173.173,Z 384.148,A -85,B 0,C 180,E1 -22979.143,E2 -22979.143} C_VEL
LIN {X 0,Y 175.89,Z 380.811,A -85,B 0,C 180,E1 -22982.962,E2 -22982.962} C_VEL
LIN {X 0,Y 178.784,Z 376.941,A -85,B 0,C 180,E1 -22986.131,E2 -22986.131} C_VEL
LIN {X 0,Y 182.947,Z 370.838,A -85,B 0,C 180,E1 -22989.803,E2 -22989.803} C_VEL
LIN {X 0,Y 187.522,Z 363.383,A -85,B 0,C 180,E1 -22993.154,E2 -22993.154} C_VEL
LIN {X 0,Y 192.167,Z 354.962,A -85,B 0,C 180,E1 -22995.987,E2 -22995.987} C_VEL
LIN {X 0,Y 194.187,Z 350.903,A -85,B 0,C 180,E1 -22997.127,E2 -22997.127} C_VEL
LIN {X 0,Y 194.839,Z 349.028,A -85,B 0,C 180,E1 -22997.683,E2 -22997.683} C_VEL
LIN {X 0,Y 195.152,Z 340.88,A -85,B 0,C 180,E1 -23000.451,E2 -23000.451} C_VEL
LIN {X 0,Y 194.461,Z 331.877,A -85,B 0,C 180,E1 -23003.414,E2 -23003.414} C_VEL
LIN {X 0,Y 193.209,Z 325.048,A -85,B 0,C 180,E1 -23005.683,E2 -23005.683} C_VEL
LIN {X 0,Y 191.055,Z 318.078,A -85,B 0,C 180,E1 -23008.179,E2 -23008.179} C_VEL
LIN {X 0,Y 187.5,Z 309.877,A -85,B 0,C 180,E1 -23011.455,E2 -23011.455} C_VEL
LIN {X 0,Y 185.775,Z 306.173,A -85,B 0,C 180,E1 -23013.005,E2 -23013.005} C_VEL
LIN {X 0,Y 183.853,Z 303.03,A -85,B 0,C 180,E1 -23014.533,E2 -23014.533} C_VEL
LIN {X 0,Y 183.332,Z 301.691,A -85,B 0,C 180,E1 -23015.062,E2 -23015.062} C_VEL
LIN {X 0,Y 180.707,Z 297.696,A -85,B 0,C 180,E1 -23017.192,E2 -23017.192} C_VEL
LIN {X 0,Y 179.952,Z 296.103,A -85,B 0,C 180,E1 -23017.923,E2 -23017.923} C_VEL
LIN {X 0,Y 177.532,Z 293.281,A -85,B 0,C 180,E1 -23019.874,E2 -23019.874} C_VEL
LIN {X 0,Y 176.404,Z 290.719,A -85,B 0,C 180,E1 -23021.065,E2 -23021.065} C_VEL
LIN {X 0,Y 173.545,Z 288.095,A -85,B 0,C 180,E1 -23023.535,E2 -23023.535} C_VEL
LIN {X 0,Y 172.2,Z 285.309,A -85,B 0,C 180,E1 -23025.073,E2 -23025.073} C_VEL
LIN {X 0,Y 172.079,Z 284.819,A -85,B 0,C 180,E1 -23025.365,E2 -23025.365} C_VEL
LIN {X 0,Y 172.161,Z 283.932,A -85,B 0,C 180,E1 -23030.605,E2 -23030.605} C_VEL
LIN {X 0,Y 172.076,Z 283.466,A -85,B 0,C 180,E1 -23035.317,E2 -23035.317} C_VEL
LIN {X 0,Y 172.514,Z 283.15,A -85,B 0,C 180,E1 -23040.003,E2 -23040.003} C_VEL
LIN {X 0,Y 172.146,Z 283.519,A -85,B 0,C 180,E1 -23047.038,E2 -23047.038} C_VEL
LIN {X 0,Y 172.124,Z 284.046,A -85,B 0,C 180,E1 -23051.502,E2 -23051.502} C_VEL
LIN {X 0,Y 172.069,Z 284.979,A -85,B 0,C 180,E1 -23056.616,E2 -23056.616} C_VEL
LIN {X 0,Y 172.227,Z 286.175,A -85,B 0,C 180,E1 -23061.549,E2 -23061.549} C_VEL
LIN {X 0,Y 172.435,Z 287.761,A -85,B 0,C 180,E1 -23066.639,E2 -23066.639} C_VEL
LIN {X 0,Y 172.534,Z 288.349,A -85,B 0,C 180,E1 -23068.184,E2 -23068.184} C_VEL
LIN {X 0,Y 173.471,Z 290.947,A -85,B 0,C 180,E1 -23069.303,E2 -23069.303} C_VEL
LIN {X 0,Y 176.178,Z 294.355,A -85,B 0,C 180,E1 -23071.743,E2 -23071.743} C_VEL
LIN {X 0,Y 177.168,Z 295.443,A -85,B 0,C 180,E1 -23072.551,E2 -23072.551} C_VEL
LIN {X 0,Y 178.981,Z 299.143,A -85,B 0,C 180,E1 -23074.275,E2 -23074.275} C_VEL
LIN {X 0,Y 180.86,Z 301.559,A -85,B 0,C 180,E1 -23075.731,E2 -23075.731} C_VEL
LIN {X 0,Y 182.952,Z 305.748,A -85,B 0,C 180,E1 -23077.553,E2 -23077.553} C_VEL
LIN {X 0,Y 184.582,Z 308.927,A -85,B 0,C 180,E1 -23078.923,E2 -23078.923} C_VEL
LIN {X 0,Y 186.551,Z 312.797,A -85,B 0,C 180,E1 -23080.535,E2 -23080.535} C_VEL
LIN {X 0,Y 190.187,Z 321.501,A -85,B 0,C 180,E1 -23083.806,E2 -23083.806} C_VEL
LIN {X 0,Y 192.342,Z 328.686,A -85,B 0,C 180,E1 -23086.194,E2 -23086.194} C_VEL
LIN {X 0,Y 193.361,Z 335.805,A -85,B 0,C 180,E1 -23088.318,E2 -23088.318} C_VEL
LIN {X 0,Y 193.583,Z 345.671,A -85,B 0,C 180,E1 -23091.174,E2 -23091.174} C_VEL
LIN {X 0,Y 192.787,Z 355.884,A -85,B 0,C 180,E1 -23094.32,E2 -23094.32} C_VEL
LIN {X 0,Y 191.793,Z 361.106,A -85,B 0,C 180,E1 -23096.027,E2 -23096.027} C_VEL
LIN {X 0,Y 187.805,Z 368.768,A -85,B 0,C 180,E1 -23098.406,E2 -23098.406} C_VEL
LIN {X 0,Y 183.372,Z 376.295,A -85,B 0,C 180,E1 -23101.375,E2 -23101.375} C_VEL
LIN {X 0,Y 179.701,Z 382.371,A -85,B 0,C 180,E1 -23104.52,E2 -23104.52} C_VEL
LIN {X 0,Y 176.408,Z 387.22,A -85,B 0,C 180,E1 -23107.761,E2 -23107.761} C_VEL
LIN {X 0,Y 173.619,Z 390.977,A -85,B 0,C 180,E1 -23111.106,E2 -23111.106} C_VEL
LIN {X 0,Y 172.123,Z 392.928,A -85,B 0,C 180,E1 -23113.393,E2 -23113.393} C_VEL
LIN {X 0,Y 171.014,Z 394.478,A -85,B 0,C 180,E1 -23115.725,E2 -23115.725} C_VEL
LIN {X 0,Y 169.483,Z 396.313,A -85,B 0,C 180,E1 -23120.453,E2 -23120.453} C_VEL
LIN {X 0,Y 168.936,Z 396.623,A -85,B 0,C 180,E1 -23125.228,E2 -23125.228} C_VEL
LIN {X 0,Y 168.914,Z 396.185,A -85,B 0,C 180,E1 -23127.616,E2 -23127.616} C_VEL
LIN {X 0,Y 169.033,Z 395.325,A -85,B 0,C 180,E1 -23130,E2 -23130} C_VEL
LIN {X 0,Y 168.909,Z 393.685,A -85,B 0,C 180,E1 -23132.991,E2 -23132.991} C_VEL
LIN {X 0,Y 169.145,Z 390.219,A -85,B 0,C 180,E1 -23137.161,E2 -23137.161} C_VEL
LIN {X 0,Y 169.673,Z 386.085,A -85,B 0,C 180,E1 -23140.742,E2 -23140.742} C_VEL
LIN {X 0,Y 170.858,Z 379.729,A -85,B 0,C 180,E1 -23144.897,E2 -23144.897} C_VEL
LIN {X 0,Y 172.662,Z 372.81,A -85,B 0,C 180,E1 -23148.388,E2 -23148.388} C_VEL
LIN {X 0,Y 173.975,Z 367.676,A -85,B 0,C 180,E1 -23150.512,E2 -23150.512} C_VEL
LIN {X 0,Y 174.481,Z 363.847,A -85,B 0,C 180,E1 -23151.961,E2 -23151.961} C_VEL
LIN {X 0,Y 173.648,Z 357.217,A -85,B 0,C 180,E1 -23154.35,E2 -23154.35} C_VEL
LIN {X 0,Y 172.292,Z 348.644,A -85,B 0,C 180,E1 -23157.089,E2 -23157.089} C_VEL
LIN {X 0,Y 172.3,Z 345.493,A -85,B 0,C 180,E1 -23157.932,E2 -23157.932} C_VEL
LIN {X 0,Y 172.544,Z 334.367,A -85,B 0,C 180,E1 -23160.549,E2 -23160.549} C_VEL
LIN {X 0,Y 172.143,Z 324.07,A -85,B 0,C 180,E1 -23162.603,E2 -23162.603} C_VEL
LIN {X 0,Y 170.822,Z 312.413,A -85,B 0,C 180,E1 -23164.625,E2 -23164.625} C_VEL
LIN {X 0,Y 168.44,Z 299.898,A -85,B 0,C 180,E1 -23166.522,E2 -23166.522} C_VEL
LIN {X 0,Y 166.391,Z 292.968,A -85,B 0,C 180,E1 -23167.539,E2 -23167.539} C_VEL
LIN {X 0,Y 165.619,Z 290.157,A -85,B 0,C 180,E1 -23167.985,E2 -23167.985} C_VEL
LIN {X 0,Y 165.092,Z 286.844,A -85,B 0,C 180,E1 -23172.93,E2 -23172.93} C_VEL
LIN {X 0,Y 164.391,Z 283.147,A -85,B 0,C 180,E1 -23178.902,E2 -23178.902} C_VEL
LIN {X 0,Y 164.327,Z 283.018,A -85,B 0,C 180,E1 -23184.349,E2 -23184.349} C_VEL
LIN {X 0,Y 164.371,Z 283.007,A -85,B 0,C 180,E1 -23189.128,E2 -23189.128} C_VEL
LIN {X 0,Y 164.395,Z 283.004,A -85,B 0,C 180,E1 -23194.688,E2 -23194.688} C_VEL
LIN {X 0,Y 164.485,Z 282.998,A -85,B 0,C 180,E1 -23200.049,E2 -23200.049} C_VEL
LIN {X 0,Y 164.503,Z 282.995,A -85,B 0,C 180,E1 -23205.144,E2 -23205.144} C_VEL
LIN {X 0,Y 164.766,Z 282.958,A -85,B 0,C 180,E1 -23210.173,E2 -23210.173} C_VEL
LIN {X 0,Y 164.828,Z 282.955,A -85,B 0,C 180,E1 -23212.648,E2 -23212.648} C_VEL
LIN {X 0,Y 165.043,Z 282.898,A -85,B 0,C 180,E1 -23217.557,E2 -23217.557} C_VEL
LIN {X 0,Y 165.293,Z 282.86,A -85,B 0,C 180,E1 -23219.997,E2 -23219.997} C_VEL
LIN {X 0,Y 164.769,Z 282.959,A -85,B 0,C 180,E1 -23224.891,E2 -23224.891} C_VEL
LIN {X 0,Y 164.85,Z 282.951,A -85,B 0,C 180,E1 -23227.345,E2 -23227.345} C_VEL
LIN {X 0,Y 164.738,Z 282.959,A -85,B 0,C 180,E1 -23231.128,E2 -23231.128} C_VEL
LIN {X 0,Y 164.476,Z 282.989,A -85,B 0,C 180,E1 -23237.401,E2 -23237.401} C_VEL
LIN {X 0,Y 164.468,Z 282.997,A -85,B 0,C 180,E1 -23239.987,E2 -23239.987} C_VEL
LIN {X 0,Y 164.382,Z 283.006,A -85,B 0,C 180,E1 -23246.128,E2 -23246.128} C_VEL
LIN {X 0,Y 164.369,Z 283.001,A -85,B 0,C 180,E1 -23251.226,E2 -23251.226} C_VEL
LIN {X 0,Y 164.343,Z 283.004,A -85,B 0,C 180,E1 -23256.773,E2 -23256.773} C_VEL
LIN {X 0,Y 164.364,Z 283.008,A -85,B 0,C 180,E1 -23259.891,E2 -23259.891} C_VEL
LIN {X 0,Y 164.332,Z 283.009,A -85,B 0,C 180,E1 -23263.363,E2 -23263.363} C_VEL
LIN {X 0,Y 164.313,Z 283.012,A -85,B 0,C 180,E1 -23266.817,E2 -23266.817} C_VEL
LIN {X 0,Y 164.298,Z 283.02,A -85,B 0,C 180,E1 -23270.346,E2 -23270.346} C_VEL
LIN {X 0,Y 164.331,Z 283.014,A -85,B 0,C 180,E1 -23274.343,E2 -23274.343} C_VEL
LIN {X 0,Y 164.363,Z 283.012,A -85,B 0,C 180,E1 -23279.13,E2 -23279.13} C_VEL
LIN {X 0,Y 164.498,Z 283.181,A -85,B 0,C 180,E1 -23284.966,E2 -23284.966} C_VEL
LIN {X 0,Y 165.661,Z 286.141,A -85,B 0,C 180,E1 -23285.452,E2 -23285.452} C_VEL
LIN {X 0,Y 169.131,Z 295.884,A -85,B 0,C 180,E1 -23287.102,E2 -23287.102} C_VEL
LIN {X 0,Y 172.174,Z 307.759,A -85,B 0,C 180,E1 -23289.225,E2 -23289.225} C_VEL
LIN {X 0,Y 173.87,Z 319.174,A -85,B 0,C 180,E1 -23291.44,E2 -23291.44} C_VEL
LIN {X 0,Y 174.689,Z 329.122,A -85,B 0,C 180,E1 -23293.643,E2 -23293.643} C_VEL
LIN {X 0,Y 174.393,Z 332.964,A -85,B 0,C 180,E1 -23294.515,E2 -23294.515} C_VEL
LIN {X 0,Y 171.705,Z 343.368,A -85,B 0,C 180,E1 -23296.99,E2 -23296.99} C_VEL
LIN {X 0,Y 169.334,Z 352.677,A -85,B 0,C 180,E1 -23299.841,E2 -23299.841} C_VEL
LIN {X 0,Y 167.214,Z 360.347,A -85,B 0,C 180,E1 -23302.756,E2 -23302.756} C_VEL
LIN {X 0,Y 165.037,Z 367.879,A -85,B 0,C 180,E1 -23306.338,E2 -23306.338} C_VEL
LIN {X 0,Y 163.599,Z 373.912,A -85,B 0,C 180,E1 -23310,E2 -23310} C_VEL
LIN {X 0,Y 162.631,Z 378.694,A -85,B 0,C 180,E1 -23313.716,E2 -23313.716} C_VEL
LIN {X 0,Y 161.889,Z 382.379,A -85,B 0,C 180,E1 -23317.483,E2 -23317.483} C_VEL
LIN {X 0,Y 161.563,Z 384.288,A -85,B 0,C 180,E1 -23320.02,E2 -23320.02} C_VEL
LIN {X 0,Y 161.468,Z 385.717,A -85,B 0,C 180,E1 -23322.569,E2 -23322.569} C_VEL
LIN {X 0,Y 161.819,Z 387.258,A -85,B 0,C 180,E1 -23327.171,E2 -23327.171} C_VEL
LIN {X 0,Y 162.291,Z 387.566,A -85,B 0,C 180,E1 -23330.269,E2 -23330.269} C_VEL
LIN {X 0,Y 163.026,Z 387.327,A -85,B 0,C 180,E1 -23332.829,E2 -23332.829} C_VEL
LIN {X 0,Y 164.35,Z 386.439,A -85,B 0,C 180,E1 -23336.11,E2 -23336.11} C_VEL
LIN {X 0,Y 166.725,Z 384.106,A -85,B 0,C 180,E1 -23340.386,E2 -23340.386} C_VEL
LIN {X 0,Y 169.338,Z 381.122,A -85,B 0,C 180,E1 -23343.902,E2 -23343.902} C_VEL
LIN {X 0,Y 172.846,Z 376.698,A -85,B 0,C 180,E1 -23347.582,E2 -23347.582} C_VEL
LIN {X 0,Y 177.396,Z 370.402,A -85,B 0,C 180,E1 -23351.374,E2 -23351.374} C_VEL
LIN {X 0,Y 181.375,Z 364.178,A -85,B 0,C 180,E1 -23354.223,E2 -23354.223} C_VEL
LIN {X 0,Y 186.044,Z 356.261,A -85,B 0,C 180,E1 -23357.02,E2 -23357.02} C_VEL
LIN {X 0,Y 188.303,Z 351.957,A -85,B 0,C 180,E1 -23358.283,E2 -23358.283} C_VEL
LIN {X 0,Y 188.979,Z 348.505,A -85,B 0,C 180,E1 -23359.495,E2 -23359.495} C_VEL
LIN {X 0,Y 189.162,Z 340.86,A -85,B 0,C 180,E1 -23362.257,E2 -23362.257} C_VEL
LIN {X 0,Y 188.484,Z 332.06,A -85,B 0,C 180,E1 -23365.349,E2 -23365.349} C_VEL
LIN {X 0,Y 187.062,Z 325.489,A -85,B 0,C 180,E1 -23367.792,E2 -23367.792} C_VEL
LIN {X 0,Y 184.892,Z 319.121,A -85,B 0,C 180,E1 -23370.39,E2 -23370.39} C_VEL
LIN {X 0,Y 181.867,Z 311.801,A -85,B 0,C 180,E1 -23373.618,E2 -23373.618} C_VEL
LIN {X 0,Y 179.677,Z 307.441,A -85,B 0,C 180,E1 -23375.754,E2 -23375.754} C_VEL
LIN {X 0,Y 176.347,Z 301.716,A -85,B 0,C 180,E1 -23378.984,E2 -23378.984} C_VEL
LIN {X 0,Y 174.191,Z 298.452,A -85,B 0,C 180,E1 -23381.096,E2 -23381.096} C_VEL
LIN {X 0,Y 173.418,Z 296.853,A -85,B 0,C 180,E1 -23382.003,E2 -23382.003} C_VEL
LIN {X 0,Y 170.928,Z 294.06,A -85,B 0,C 180,E1 -23384.502,E2 -23384.502} C_VEL
LIN {X 0,Y 169.635,Z 291.347,A -85,B 0,C 180,E1 -23386.221,E2 -23386.221} C_VEL
LIN {X 0,Y 166.76,Z 288.759,A -85,B 0,C 180,E1 -23389.643,E2 -23389.643} C_VEL
